// TIA Portal project "HydroPlantProject" (V15)

(* hardware
DEVICE "S71500/ET200MP station_1"  S7-1500 station
   slot 0: "Rail_0"  Rack  6ES7 590-1***0-0AA0
   slot 1: "PLC_1"  CPU 1511-1 PN  6ES7 511-1AK00-0AB0  V1.8
      slot 3: "CPU display_1"  6ES7591-1AA00-0AA0
DEVICE "PC-System_1"  SIMATIC PC station
   slot 0: "SIMATIC PC station"  Rail  SIMATIC PC-Station  V1.0
      slot 125: "Stationmanager"  Station_Manager  V6.0.4
   slot 1: "HMI_RT_1"  WinCC RT Advanced  6AV2 104-0xxxx-xxxx  15.0.0.0
      slot 33792: "Host interface"  Host interface
   slot 2: "IE general_1"  IE General  IE_CP  V8.2.0
*)

// ===== PLC "PLC_1"  CPU 1511-1 PN =====

VAR_GLOBAL   // PLC tag table "Default tag table"
   "Brake_Out" AT %M0.0 : Bool;
   "Baffle_Out" AT %MW18 : Int;
   "RPM_In" AT %MW2 : Int;
   "OilTemp_In" AT %MW4 : Int;
   "OilPumpVFDen_Out" AT %M0.1 : Bool;
   "OilPumpVFDsp_Out" AT %MW6 : Int;
   "OilFlow_In" AT %MW8 : Int;
   "Current_In" AT %MW10 : Int;
   "Baffle_En" AT %M0.2 : Bool;
   "ProgLang" AT %MW12 : Int;
   "ONS1" AT %M0.3 : Bool;
   "PB_LAD" AT %M0.4 : Bool;
   "ONS" AT %M0.5 : Bool;
   "PB_FBD" AT %M0.6 : Bool;
   "PB_SCL" AT %M0.7 : Bool;
   "PB_STL" AT %M1.0 : Bool;
   "ONS2" AT %M1.1 : Bool;
   "ONS3" AT %M1.2 : Bool;
   "ONS4" AT %M1.3 : Bool;
   "AlarmHorn_Out" AT %M1.4 : Bool;
   "Stationinterlock_Out" AT %M1.5 : Bool;
   "OilPumpVFDpct" AT %MW14 : Int;
   "BafflePct" AT %MW16 : Int;
   "OilTemp" AT %MW20 : Int;
   "OilFlow" AT %MW24 : Int;
   "RPM" AT %MW26 : Int;
   "Current" AT %MW28 : Int;
   "OilPumpVFDhand_Pb" AT %M1.6 : Bool;
   "OilPumpVFDoff_Pb" AT %M1.7 : Bool;
   "OilPumpVFDauto_Pb" AT %M22.0 : Bool;
   "OilPumpVFDhoa" AT %MW30 : Int;
   "BrakeHoa" AT %MW32 : Int;
   "BrakeOff_Pb" AT %M22.1 : Bool;
   "BrakeHand_Pb" AT %M22.2 : Bool;
   "BrakeAuto_Pb" AT %M22.3 : Bool;
   "AlarmHornOff_Pb" AT %M22.4 : Bool;
   "AlarmHornHand_Pb" AT %M22.5 : Bool;
   "AlarmHornHoa" AT %MW34 : Int;
   "AlarmHornAuto_Pb" AT %M22.6 : Bool;
   "StationintOff_Pb" AT %M22.7 : Bool;
   "StationintHand_Pb" AT %M23.0 : Bool;
   "StationintAuto_Pb" AT %M23.1 : Bool;
   "StationintHoa" AT %MW36 : Int;
   "OilPumpVFD_Ctrl" AT %M23.2 : Bool;
   "Bracke_Ctrl" AT %M23.3 : Bool;
   "ALarmHorn_Ctrl" AT %M23.4 : Bool;
   "Stationint_Ctrl" AT %M23.5 : Bool;
   "OilLowFlowDelay_Sp" AT %MW38 : Int;
   "AlarmReset" AT %M23.6 : Bool;
   "AlarmSilence" AT %M23.7 : Bool;
   "OilLowFlowAlarm" AT %M40.0 : Bool;
   "OilLowFlowNotify" AT %M40.1 : Bool;
   "OilLLFlow_Sp" AT %MW42 : Int;
   "OverCurrent_Sp" AT %MW44 : Int;
   "OverCurrentAlarm" AT %M40.2 : Bool;
   "OverCurrentAlarm(1)" AT %M40.3 : Bool;
   "OverCurrentNotify" AT %M40.4 : Bool;
   "OverCurrentDelay_Sp" AT %MW46 : Int;
   "HighoilTepDelay_Sp" AT %MW48 : Int;
   "HighOilTemp _Sp" AT %MW50 : Int;
   "OilTempAlarm" AT %M40.5 : Bool;
   "OilTempAlarmNotify" AT %M40.6 : Bool;
   "RottorOverspeed_Sp" AT %MW52 : Int;
   "RottorOverspeedDelay_Sp" AT %MW54 : Int;
   "RottorOverspeedAlarm" AT %M40.7 : Bool;
   "RottorOverspeedNotify" AT %M41.0 : Bool;
   "OilHighFlowAlarm" AT %M41.1 : Bool;
   "OilHighFlowNotify" AT %M41.2 : Bool;
   "OilHighFlowDelay_Sp" AT %MW56 : Int;
   "OilHHFlow_Sp" AT %MW58 : Int;
   "BraheFailuerDelay_Sp" AT %MW60 : Int;
   "BrakeFalierAlarm" AT %M41.3 : Bool;
   "BrakeFalierAlarmNotify" AT %M41.4 : Bool;
   "EStop" AT %M41.5 : Bool;
   "ESTOPAlarm" AT %M41.6 : Bool;
   "EStapAlarmNotify" AT %M41.7 : Bool;
   "Tag_1" AT %T1 : Timer;
   "WarmupMode" AT %M62.0 : Bool;
   "StabilizeMode" AT %M62.1 : Bool;
   "GenerationMode" AT %M62.2 : Bool;
   "CooldownMode" AT %M62.3 : Bool;
   "IdleMode" AT %M62.4 : Bool;
   "FaultMode" AT %M62.5 : Bool;
   "SystemSTART_Pb" AT %M62.6 : Bool;
   "WarmupRPM" AT %MW63 : Int;
   "RPM_SP" AT %MW64 : Int;
   "BaffleHOA" AT %MW66 : Int;
   "Baffle_Ctrl" AT %M62.7 : Bool;
   "WarmupVFDpct" AT %MW68 : Int;
   "VFD_sp" AT %MW70 : Int;
   "WarmupOILTemp" AT %MW72 : Int;
   "WarmupOilTempDelay_sp" AT %MW74 : Int;
   "WarmupTransition" AT %M76.0 : Bool;
   "BafflePIDsp" AT %MW78 : Int;
   "StabilizeKWsp" AT %MW80 : Int;
   "StabilizeDelay_sp" AT %MW82 : Int;
   "StabilizeTranzition" AT %M76.1 : Bool;
   "STARTSequnceBIT" AT %M76.2 : Bool;
   "SystemSTOP_PB" AT %M76.3 : Bool;
   "GenerationTransition" AT %M76.4 : Bool;
   "BafflePIDin" AT %MW84 : Int;
   "CooldownRPM" AT %MW86 : Int;
   "CooldownDelay_Sp" AT %MW88 : Int;
   "CooldawnTransition" AT %M76.5 : Bool;
   "CoolDownRPM_sp" AT %MW90 : Int;
   "CoolDownOilTemp_sp" AT %MW92 : Int;
   "SequenceRunning" AT %M76.6 : Bool;
   "ONS5" AT %M76.7 : Bool;
   "StabilizeTransition" AT %M77.0 : Bool;
END_VAR

DATA_BLOCK "SimLogic_DB"   // DB1
{ S7_Optimized_Access := 'TRUE' }
VERSION : 0.1
// stored: InstanceOfName SimLogic
"SimLogic"
BEGIN
END_DATA_BLOCK

DATA_BLOCK "SimLogic_DB_1"   // DB2
{ S7_Optimized_Access := 'TRUE' }
VERSION : 0.1
// stored: InstanceOfName SimLogic
"SimLogic"
BEGIN
END_DATA_BLOCK

DATA_BLOCK "IO_LAD_DB"   // DB4
{ S7_Optimized_Access := 'TRUE' }
VERSION : 0.1
// stored: InstanceOfName IO_LAD
"IO_LAD"
BEGIN
END_DATA_BLOCK

DATA_BLOCK "IO_FBD_DB"   // DB5
{ S7_Optimized_Access := 'TRUE' }
VERSION : 0.1
// stored: InstanceOfName IO_FBD
"IO_FBD"
BEGIN
END_DATA_BLOCK

DATA_BLOCK "IO_SCL_DB"   // DB6
{ S7_Optimized_Access := 'TRUE' }
VERSION : 0.1
// stored: InstanceOfName IO_SCL
"IO_SCL"
BEGIN
END_DATA_BLOCK

DATA_BLOCK "IO_STL_DB"   // DB7
{ S7_Optimized_Access := 'TRUE' }
VERSION : 0.1
// stored: InstanceOfName IO_STL
"IO_STL"
BEGIN
END_DATA_BLOCK

DATA_BLOCK "ALARMS_LAD_DB"   // DB8
{ S7_Optimized_Access := 'TRUE' }
VERSION : 0.1
// stored: InstanceOfName ALARMS_LAD
"ALARMS_LAD"
BEGIN
END_DATA_BLOCK

DATA_BLOCK "SCP_DB"   // DB9
{ S7_Optimized_Access := 'TRUE' }
VERSION : 0.1
// stored: InstanceOfName SCP
"SCP"
BEGIN
END_DATA_BLOCK

DATA_BLOCK "SCP_DB_1"   // DB10
{ S7_Optimized_Access := 'TRUE' }
VERSION : 0.1
// stored: InstanceOfName SCP
"SCP"
BEGIN
END_DATA_BLOCK

DATA_BLOCK "HOA_LAD_DB"   // DB11
{ S7_Optimized_Access := 'TRUE' }
VERSION : 0.1
// stored: InstanceOfName HOA_LAD
"HOA_LAD"
BEGIN
END_DATA_BLOCK

DATA_BLOCK "HOA_FBD_DB"   // DB12
{ S7_Optimized_Access := 'TRUE' }
VERSION : 0.1
// stored: InstanceOfName HOA_FBD
"HOA_FBD"
BEGIN
END_DATA_BLOCK

DATA_BLOCK "HOA_SCL_DB"   // DB13
{ S7_Optimized_Access := 'TRUE' }
VERSION : 0.1
// stored: InstanceOfName HOA_SCL
"HOA_SCL"
BEGIN
END_DATA_BLOCK

DATA_BLOCK "HOA_STL_DB"   // DB14
{ S7_Optimized_Access := 'TRUE' }
VERSION : 0.1
// stored: InstanceOfName HOA_STL
"HOA_STL"
BEGIN
END_DATA_BLOCK

DATA_BLOCK "ALARMS_FBD_DB"   // DB15
{ S7_Optimized_Access := 'TRUE' }
VERSION : 0.1
// stored: InstanceOfName ALARMS_FBD
"ALARMS_FBD"
BEGIN
END_DATA_BLOCK

DATA_BLOCK "ALARMS_SCL_DB"   // DB16
{ S7_Optimized_Access := 'TRUE' }
VERSION : 0.1
// stored: InstanceOfName ALARMS_SCL
"ALARMS_SCL"
BEGIN
END_DATA_BLOCK

DATA_BLOCK "ALARMS_STL_DB"   // DB18
{ S7_Optimized_Access := 'TRUE' }
VERSION : 0.1
// stored: InstanceOfName ALARMS_STL
"ALARMS_STL"
BEGIN
END_DATA_BLOCK

DATA_BLOCK "SEQUENCE_DB"   // DB37
{ S7_Optimized_Access := 'TRUE' }
VERSION : 0.1
// stored: InstanceOfName SEQUENCE
"SEQUENCE"
BEGIN
END_DATA_BLOCK

// folder: System blocks/Program resources

DATA_BLOCK "IEC_Timer_0_DB_25"   // DB3
{ S7_Optimized_Access := 'TRUE' }
AUTHOR : Simatic
FAMILY : IEC
NAME : IEC_TMR
VERSION : 1.0
// stored: InstanceOfName IEC_TIMER
"IEC_TIMER"
BEGIN
END_DATA_BLOCK

DATA_BLOCK "IEC_Timer_0_DB"   // DB17
{ S7_Optimized_Access := 'TRUE' }
AUTHOR : Simatic
FAMILY : IEC
NAME : IEC_TMR
VERSION : 1.0
// stored: InstanceOfName IEC_TIMER
"IEC_TIMER"
BEGIN
END_DATA_BLOCK

DATA_BLOCK "IEC_Timer_0_DB_1"   // DB19
{ S7_Optimized_Access := 'TRUE' }
AUTHOR : Simatic
FAMILY : IEC
NAME : IEC_TMR
VERSION : 1.0
// stored: InstanceOfName IEC_TIMER
"IEC_TIMER"
BEGIN
END_DATA_BLOCK

DATA_BLOCK "IEC_Timer_0_DB_2"   // DB20
{ S7_Optimized_Access := 'TRUE' }
AUTHOR : Simatic
FAMILY : IEC
NAME : IEC_TMR
VERSION : 1.0
// stored: InstanceOfName IEC_TIMER
"IEC_TIMER"
BEGIN
END_DATA_BLOCK

DATA_BLOCK "IEC_Timer_0_DB_3"   // DB21
{ S7_Optimized_Access := 'TRUE' }
AUTHOR : Simatic
FAMILY : IEC
NAME : IEC_TMR
VERSION : 1.0
// stored: InstanceOfName IEC_TIMER
"IEC_TIMER"
BEGIN
END_DATA_BLOCK

DATA_BLOCK "IEC_Timer_0_DB_4"   // DB22
{ S7_Optimized_Access := 'TRUE' }
AUTHOR : Simatic
FAMILY : IEC
NAME : IEC_TMR
VERSION : 1.0
// stored: InstanceOfName IEC_TIMER
"IEC_TIMER"
BEGIN
END_DATA_BLOCK

DATA_BLOCK "IEC_Timer_0_DB_5"   // DB23
{ S7_Optimized_Access := 'TRUE' }
AUTHOR : Simatic
FAMILY : IEC
NAME : IEC_TMR
VERSION : 1.0
// stored: InstanceOfName IEC_TIMER
"IEC_TIMER"
BEGIN
END_DATA_BLOCK

DATA_BLOCK "IEC_Timer_0_DB_6"   // DB24
{ S7_Optimized_Access := 'TRUE' }
AUTHOR : Simatic
FAMILY : IEC
NAME : IEC_TMR
VERSION : 1.0
// stored: InstanceOfName IEC_TIMER
"IEC_TIMER"
BEGIN
END_DATA_BLOCK

DATA_BLOCK "IEC_Timer_0_DB_7"   // DB25
{ S7_Optimized_Access := 'TRUE' }
AUTHOR : Simatic
FAMILY : IEC
NAME : IEC_TMR
VERSION : 1.0
// stored: InstanceOfName IEC_TIMER
"IEC_TIMER"
BEGIN
END_DATA_BLOCK

DATA_BLOCK "IEC_Timer_0_DB_8"   // DB26
{ S7_Optimized_Access := 'TRUE' }
AUTHOR : Simatic
FAMILY : IEC
NAME : IEC_TMR
VERSION : 1.0
// stored: InstanceOfName IEC_TIMER
"IEC_TIMER"
BEGIN
END_DATA_BLOCK

DATA_BLOCK "IEC_Timer_0_DB_9"   // DB27
{ S7_Optimized_Access := 'TRUE' }
AUTHOR : Simatic
FAMILY : IEC
NAME : IEC_TMR
VERSION : 1.0
// stored: InstanceOfName IEC_TIMER
"IEC_TIMER"
BEGIN
END_DATA_BLOCK

DATA_BLOCK "IEC_Timer_0_DB_10"   // DB28
{ S7_Optimized_Access := 'TRUE' }
AUTHOR : Simatic
FAMILY : IEC
NAME : IEC_TMR
VERSION : 1.0
// stored: InstanceOfName IEC_TIMER
"IEC_TIMER"
BEGIN
END_DATA_BLOCK

DATA_BLOCK "IEC_Timer_0_DB_11"   // DB29
{ S7_Optimized_Access := 'TRUE' }
AUTHOR : Simatic
FAMILY : IEC
NAME : IEC_TMR
VERSION : 1.0
// stored: InstanceOfName IEC_TIMER
"IEC_TIMER"
BEGIN
END_DATA_BLOCK

DATA_BLOCK "IEC_Timer_0_DB_12"   // DB30
{ S7_Optimized_Access := 'TRUE' }
AUTHOR : Simatic
FAMILY : IEC
NAME : IEC_TMR
VERSION : 1.0
// stored: InstanceOfName IEC_TIMER
"IEC_TIMER"
BEGIN
END_DATA_BLOCK

DATA_BLOCK "IEC_Timer_0_DB_13"   // DB31
{ S7_Optimized_Access := 'TRUE' }
AUTHOR : Simatic
FAMILY : IEC
NAME : IEC_TMR
VERSION : 1.0
// stored: InstanceOfName IEC_TIMER
"IEC_TIMER"
BEGIN
END_DATA_BLOCK

DATA_BLOCK "IEC_Timer_0_DB_14"   // DB32
{ S7_Optimized_Access := 'TRUE' }
AUTHOR : Simatic
FAMILY : IEC
NAME : IEC_TMR
VERSION : 1.0
// stored: InstanceOfName IEC_TIMER
"IEC_TIMER"
BEGIN
END_DATA_BLOCK

DATA_BLOCK "IEC_Timer_0_DB_15"   // DB33
{ S7_Optimized_Access := 'TRUE' }
AUTHOR : Simatic
FAMILY : IEC
NAME : IEC_TMR
VERSION : 1.0
// stored: InstanceOfName IEC_TIMER
"IEC_TIMER"
BEGIN
END_DATA_BLOCK

DATA_BLOCK "IEC_Timer_0_DB_16"   // DB34
{ S7_Optimized_Access := 'TRUE' }
AUTHOR : Simatic
FAMILY : IEC
NAME : IEC_TMR
VERSION : 1.0
// stored: InstanceOfName IEC_TIMER
"IEC_TIMER"
BEGIN
END_DATA_BLOCK

DATA_BLOCK "IEC_Timer_0_DB_17"   // DB35
{ S7_Optimized_Access := 'TRUE' }
AUTHOR : Simatic
FAMILY : IEC
NAME : IEC_TMR
VERSION : 1.0
// stored: InstanceOfName IEC_TIMER
"IEC_TIMER"
BEGIN
END_DATA_BLOCK

DATA_BLOCK "IEC_Timer_0_DB_18"   // DB36
{ S7_Optimized_Access := 'TRUE' }
AUTHOR : Simatic
FAMILY : IEC
NAME : IEC_TMR
VERSION : 1.0
// stored: InstanceOfName IEC_TIMER
"IEC_TIMER"
BEGIN
END_DATA_BLOCK

DATA_BLOCK "IEC_Timer_0_DB_19"   // DB38
{ S7_Optimized_Access := 'TRUE' }
AUTHOR : Simatic
FAMILY : IEC
NAME : IEC_TMR
VERSION : 1.0
// stored: InstanceOfName IEC_TIMER
"IEC_TIMER"
BEGIN
END_DATA_BLOCK

DATA_BLOCK "IEC_Timer_0_DB_20"   // DB39
{ S7_Optimized_Access := 'TRUE' }
AUTHOR : Simatic
FAMILY : IEC
NAME : IEC_TMR
VERSION : 1.0
// stored: InstanceOfName IEC_TIMER
"IEC_TIMER"
BEGIN
END_DATA_BLOCK

DATA_BLOCK "IEC_Timer_0_DB_30"   // DB40
{ S7_Optimized_Access := 'TRUE' }
AUTHOR : Simatic
FAMILY : IEC
NAME : IEC_TMR
VERSION : 1.0
// stored: InstanceOfName IEC_TIMER
"IEC_TIMER"
BEGIN
END_DATA_BLOCK

DATA_BLOCK "IEC_Timer_0_DB_21"   // DB41
{ S7_Optimized_Access := 'TRUE' }
AUTHOR : Simatic
FAMILY : IEC
NAME : IEC_TMR
VERSION : 1.0
// stored: InstanceOfName IEC_TIMER
"IEC_TIMER"
BEGIN
END_DATA_BLOCK

DATA_BLOCK "IEC_Timer_1_DB"   // DB43
{ S7_Optimized_Access := 'TRUE' }
AUTHOR : Simatic
FAMILY : IEC
NAME : IEC_TMR
VERSION : 1.0
// stored: InstanceOfName IEC_TIMER
"IEC_TIMER"
BEGIN
END_DATA_BLOCK

DATA_BLOCK "IEC_Timer_0_DB_22"   // DB44
{ S7_Optimized_Access := 'TRUE' }
AUTHOR : Simatic
FAMILY : IEC
NAME : IEC_TMR
VERSION : 1.0
// stored: InstanceOfName IEC_TIMER
"IEC_TIMER"
BEGIN
END_DATA_BLOCK

DATA_BLOCK "IEC_Timer_0_DB_23"   // DB45
{ S7_Optimized_Access := 'TRUE' }
AUTHOR : Simatic
FAMILY : IEC
NAME : IEC_TMR
VERSION : 1.0
// stored: InstanceOfName IEC_TIMER
"IEC_TIMER"
BEGIN
END_DATA_BLOCK

DATA_BLOCK "IEC_Timer_0_DB_24"   // DB46
{ S7_Optimized_Access := 'TRUE' }
AUTHOR : Simatic
FAMILY : IEC
NAME : IEC_TMR
VERSION : 1.0
// stored: InstanceOfName IEC_TIMER
"IEC_TIMER"
BEGIN
END_DATA_BLOCK

DATA_BLOCK "IEC_Timer_0_DB_26"   // DB47
{ S7_Optimized_Access := 'TRUE' }
AUTHOR : Simatic
FAMILY : IEC
NAME : IEC_TMR
VERSION : 1.0
// stored: InstanceOfName IEC_TIMER
"IEC_TIMER"
BEGIN
END_DATA_BLOCK

DATA_BLOCK "IEC_Timer_0_DB_27"   // DB48
{ S7_Optimized_Access := 'TRUE' }
AUTHOR : Simatic
FAMILY : IEC
NAME : IEC_TMR
VERSION : 1.0
// stored: InstanceOfName IEC_TIMER
"IEC_TIMER"
BEGIN
END_DATA_BLOCK

// folder: (top level)

FUNCTION_BLOCK "SimLogic"   // FB1, FBD
{ S7_Optimized_Access := 'TRUE' }
VERSION : 0.1
   VAR
      "TO" : Bool;
      rpmv : Int;
      addrpmv : Bool;
      otsp : Int;
      ott : Int;
      TO1 : Bool;
      TO2 : Bool;
      be2 : Int;
      be3 : Int;
      be1 : Int;
      TO3 : Bool;
   END_VAR
   VAR_TEMP
      bf : Int;
      rpmvt : Int;
      bfr : Real;
   END_VAR
BEGIN

REGION Network 1
   // RPM
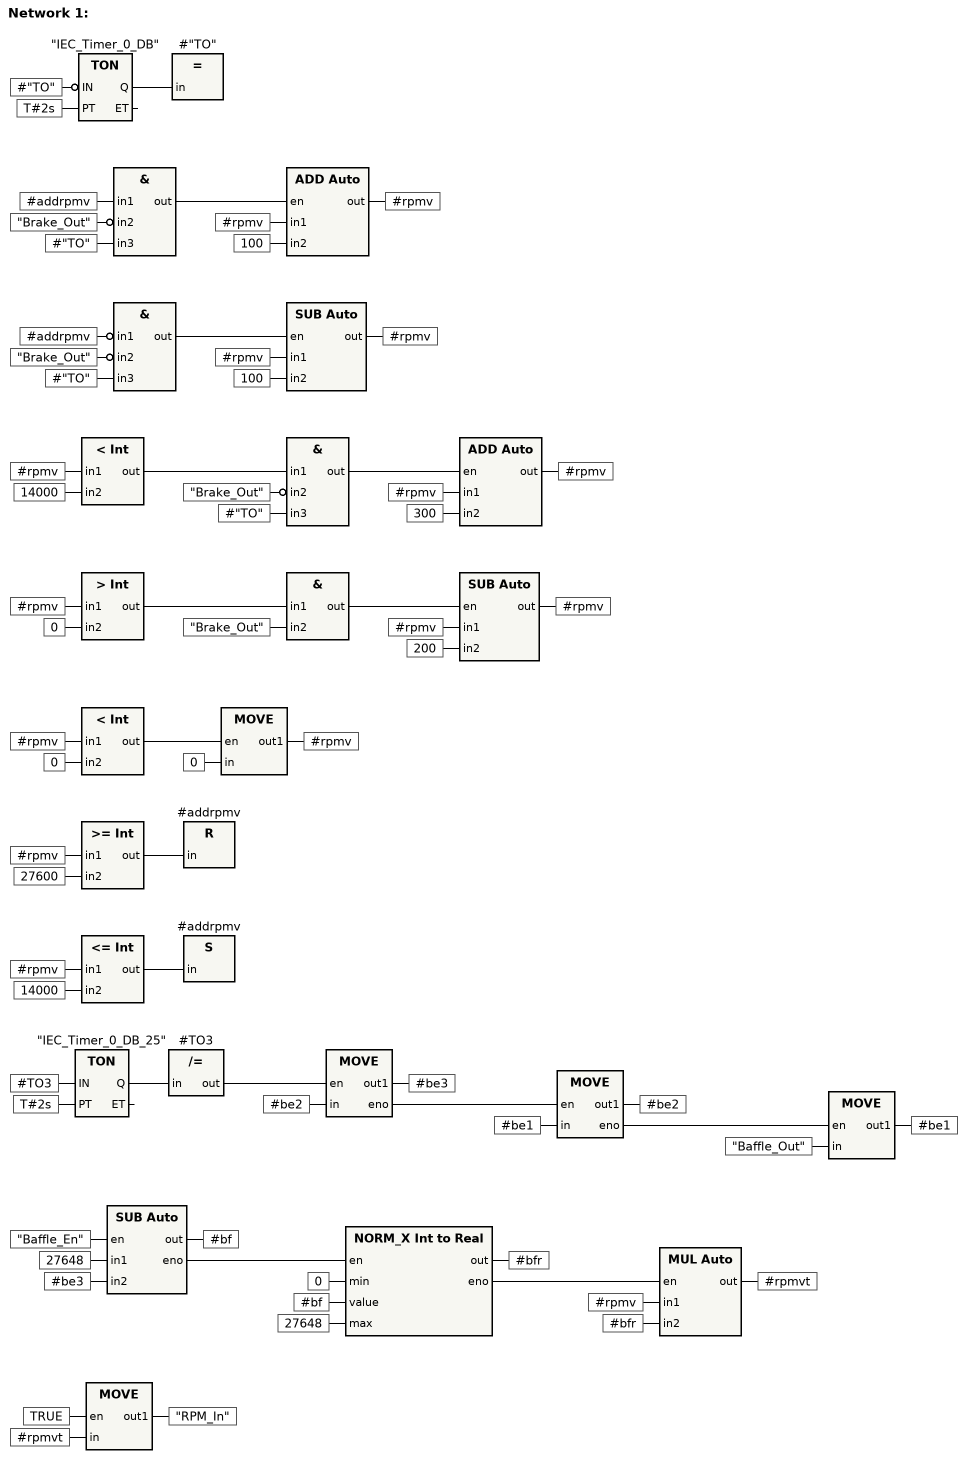
   "IEC_Timer_0_DB".TON(IN := NOT #"TO", PT := T#2s);
   #"TO" := "IEC_Timer_0_DB".Q;
   IF #addrpmv AND NOT "Brake_Out" AND #"TO" THEN #rpmv := #rpmv + 100; END_IF;
   IF NOT #addrpmv AND NOT "Brake_Out" AND #"TO" THEN #rpmv := #rpmv - 100; END_IF;
   IF (#rpmv < 14000) AND NOT "Brake_Out" AND #"TO" THEN #rpmv := #rpmv + 300; END_IF;
   IF (#rpmv > 0) AND "Brake_Out" THEN #rpmv := #rpmv - 200; END_IF;
   IF #rpmv < 0 THEN #rpmv := 0; END_IF;
   IF #rpmv >= 27600 THEN #addrpmv := FALSE; END_IF;
   IF #rpmv <= 14000 THEN #addrpmv := TRUE; END_IF;
   "IEC_Timer_0_DB_25".TON(IN := #TO3, PT := T#2s);
   #TO3 := NOT "IEC_Timer_0_DB_25".Q;
   IF "IEC_Timer_0_DB_25".Q THEN
       #be3 := #be2;
       #be2 := #be1;
       #be1 := "Baffle_Out";
   END_IF;
   IF "Baffle_En" THEN
       #bf := 27648 - #be3;
       #bfr := NORM_X(MIN := 0, VALUE := #bf, MAX := 27648);
       #rpmvt := #rpmv * #bfr;
   END_IF;
   IF TRUE THEN "RPM_In" := #rpmvt; END_IF;
END_REGION

REGION Network 2
   // Oil Temp
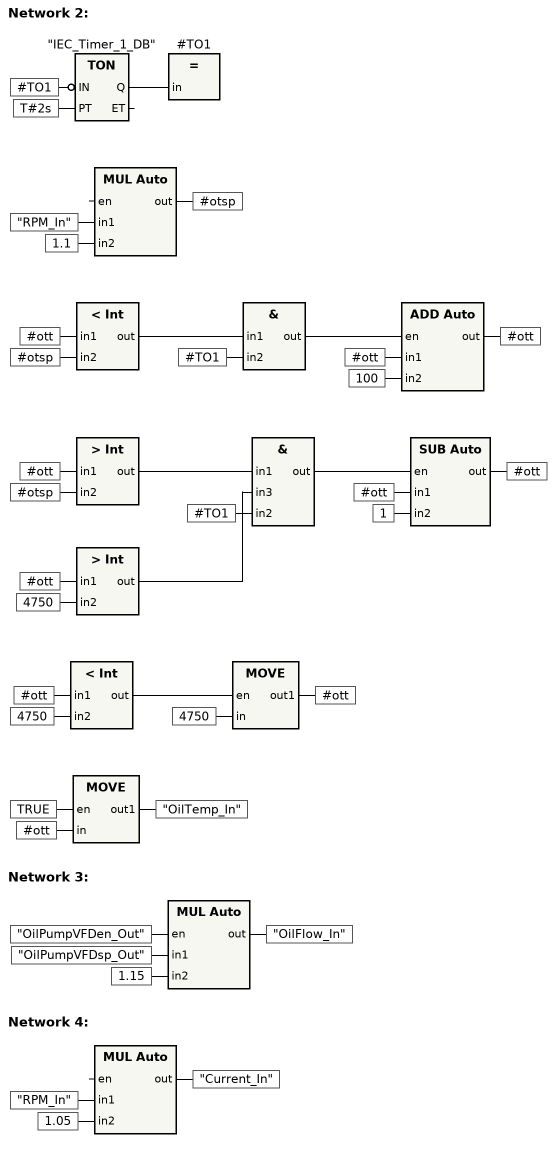
   "IEC_Timer_1_DB".TON(IN := NOT #TO1, PT := T#2s);
   #TO1 := "IEC_Timer_1_DB".Q;
   #otsp := "RPM_In" * 1.1;
   IF (#ott < #otsp) AND #TO1 THEN #ott := #ott + 100; END_IF;
   IF (#ott > #otsp) AND (#ott > 4750) AND #TO1 THEN #ott := #ott - 1; END_IF;
   IF #ott < 4750 THEN #ott := 4750; END_IF;
   IF TRUE THEN "OilTemp_In" := #ott; END_IF;
END_REGION

REGION Network 3
   // Oil Flow
   IF "OilPumpVFDen_Out" THEN "OilFlow_In" := "OilPumpVFDsp_Out" * 1.15; END_IF;
END_REGION

REGION Network 4
   // Current
   "Current_In" := "RPM_In" * 1.05;
END_REGION
END_FUNCTION_BLOCK

FUNCTION_BLOCK "IO_LAD"   // FB2, LAD
{ S7_Optimized_Access := 'TRUE' }
VERSION : 0.1
BEGIN

REGION Network 1
   // Digital Output
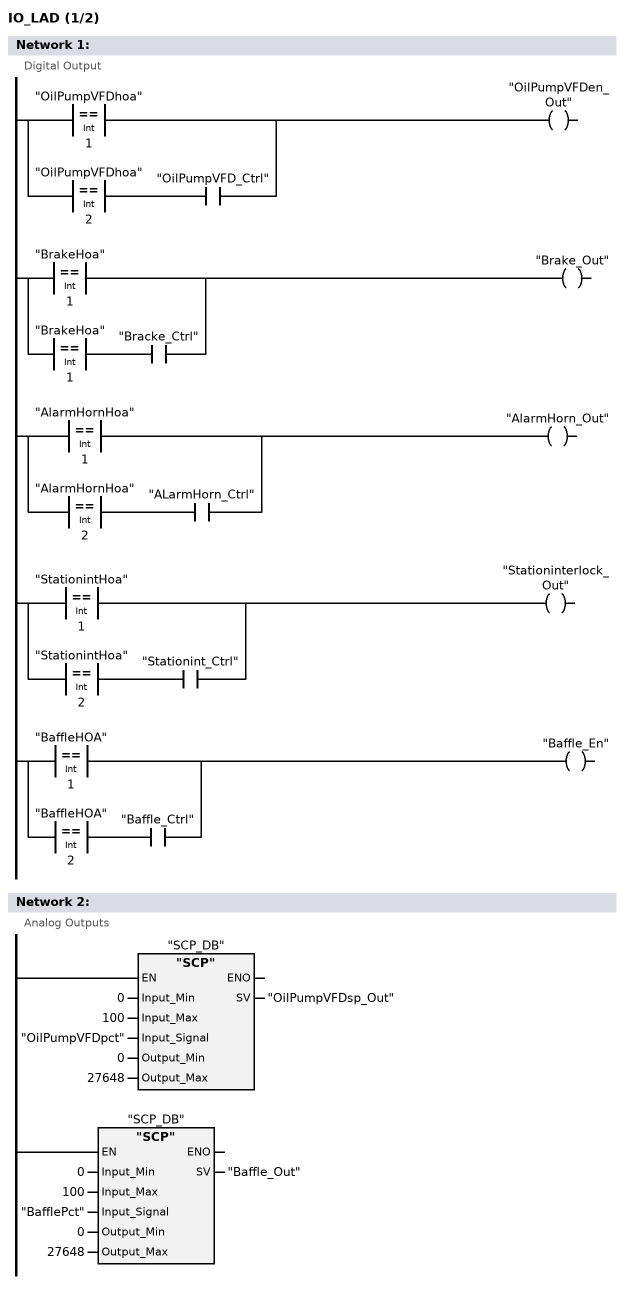
   RUNG wire#powerrail
      { S7_Templates := "SrcType := Int" } EQ_Contact(in1 := "OilPumpVFDhoa", in2 := 1)
      wire#w1
      Coil( "OilPumpVFDen_Out" )
   END_RUNG
   RUNG wire#powerrail
      { S7_Templates := "SrcType := Int" } EQ_Contact(in1 := "OilPumpVFDhoa", in2 := 2)
      Contact( "OilPumpVFD_Ctrl" )
   END_RUNG wire#w1
   RUNG wire#powerrail
      { S7_Templates := "SrcType := Int" } EQ_Contact(in1 := "BrakeHoa", in2 := 1)
      wire#w2
      Coil( "Brake_Out" )
   END_RUNG
   RUNG wire#powerrail
      { S7_Templates := "SrcType := Int" } EQ_Contact(in1 := "BrakeHoa", in2 := 1)
      Contact( "Bracke_Ctrl" )
   END_RUNG wire#w2
   RUNG wire#powerrail
      { S7_Templates := "SrcType := Int" } EQ_Contact(in1 := "AlarmHornHoa", in2 := 1)
      wire#w3
      Coil( "AlarmHorn_Out" )
   END_RUNG
   RUNG wire#powerrail
      { S7_Templates := "SrcType := Int" } EQ_Contact(in1 := "AlarmHornHoa", in2 := 2)
      Contact( "ALarmHorn_Ctrl" )
   END_RUNG wire#w3
   RUNG wire#powerrail
      { S7_Templates := "SrcType := Int" } EQ_Contact(in1 := "StationintHoa", in2 := 1)
      wire#w4
      Coil( "Stationinterlock_Out" )
   END_RUNG
   RUNG wire#powerrail
      { S7_Templates := "SrcType := Int" } EQ_Contact(in1 := "StationintHoa", in2 := 2)
      Contact( "Stationint_Ctrl" )
   END_RUNG wire#w4
   RUNG wire#powerrail
      { S7_Templates := "SrcType := Int" } EQ_Contact(in1 := "BaffleHOA", in2 := 1)
      wire#w5
      Coil( "Baffle_En" )
   END_RUNG
   RUNG wire#powerrail
      { S7_Templates := "SrcType := Int" } EQ_Contact(in1 := "BaffleHOA", in2 := 2)
      Contact( "Baffle_Ctrl" )
   END_RUNG wire#w5
   // the same network as SCL:
   "OilPumpVFDen_Out" := ("OilPumpVFDhoa" = 1) OR (("OilPumpVFDhoa" = 2) AND "OilPumpVFD_Ctrl");
   "Brake_Out" := ("BrakeHoa" = 1) OR (("BrakeHoa" = 1) AND "Bracke_Ctrl");
   "AlarmHorn_Out" := ("AlarmHornHoa" = 1) OR (("AlarmHornHoa" = 2) AND "ALarmHorn_Ctrl");
   "Stationinterlock_Out" := ("StationintHoa" = 1) OR (("StationintHoa" = 2) AND "Stationint_Ctrl");
   "Baffle_En" := ("BaffleHOA" = 1) OR (("BaffleHOA" = 2) AND "Baffle_Ctrl");
END_REGION

REGION Network 2
   // Analog Outputs
   RUNG wire#powerrail
      "SCP_DB"(Input_Min := 0, Input_Max := 100, Input_Signal := "OilPumpVFDpct", Output_Min := 0, Output_Max := 27648, SV => "OilPumpVFDsp_Out")
   END_RUNG
   RUNG wire#powerrail
      "SCP_DB"(Input_Min := 0, Input_Max := 100, Input_Signal := "BafflePct", Output_Min := 0, Output_Max := 27648, SV => "Baffle_Out")
   END_RUNG
   // the same network as SCL:
   "SCP_DB"(Input_Min := 0,   // "SCP"
            Input_Max := 100,
            Input_Signal := "OilPumpVFDpct",
            Output_Min := 0,
            Output_Max := 27648,
            SV => "OilPumpVFDsp_Out");
   "SCP_DB"(Input_Min := 0,   // "SCP"
            Input_Max := 100,
            Input_Signal := "BafflePct",
            Output_Min := 0,
            Output_Max := 27648,
            SV => "Baffle_Out");
END_REGION

REGION Network 3
   // Analog Inputs
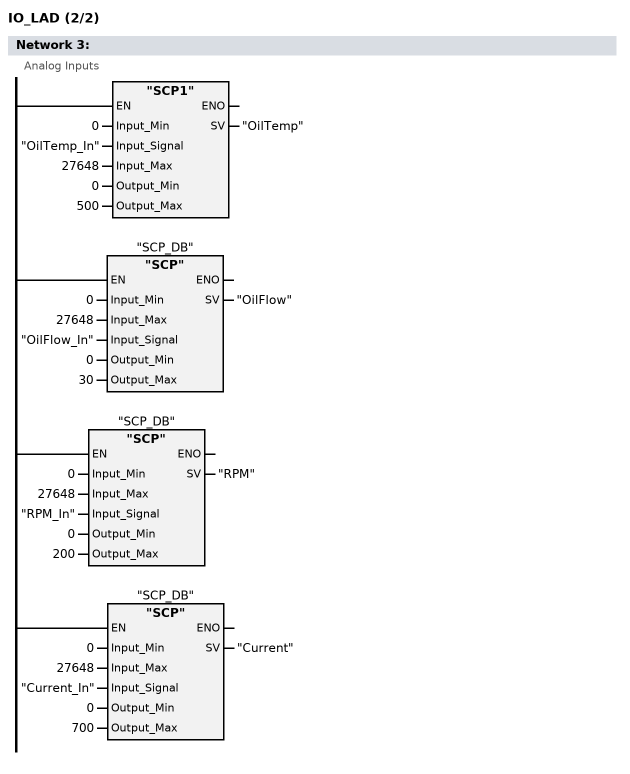
   RUNG wire#powerrail
      "SCP1"(Input_Min := 0, Input_Signal := "OilTemp_In", Input_Max := 27648, Output_Min := 0, Output_Max := 500, SV => "OilTemp")
   END_RUNG
   RUNG wire#powerrail
      "SCP_DB"(Input_Min := 0, Input_Max := 27648, Input_Signal := "OilFlow_In", Output_Min := 0, Output_Max := 30, SV => "OilFlow")
   END_RUNG
   RUNG wire#powerrail
      "SCP_DB"(Input_Min := 0, Input_Max := 27648, Input_Signal := "RPM_In", Output_Min := 0, Output_Max := 200, SV => "RPM")
   END_RUNG
   RUNG wire#powerrail
      "SCP_DB"(Input_Min := 0, Input_Max := 27648, Input_Signal := "Current_In", Output_Min := 0, Output_Max := 700, SV => "Current")
   END_RUNG
   // the same network as SCL:
   "SCP1"(Input_Min := 0,
          Input_Signal := "OilTemp_In",
          Input_Max := 27648,
          Output_Min := 0,
          Output_Max := 500,
          SV => "OilTemp");
   "SCP_DB"(Input_Min := 0,   // "SCP"
            Input_Max := 27648,
            Input_Signal := "OilFlow_In",
            Output_Min := 0,
            Output_Max := 30,
            SV => "OilFlow");
   "SCP_DB"(Input_Min := 0,   // "SCP"
            Input_Max := 27648,
            Input_Signal := "RPM_In",
            Output_Min := 0,
            Output_Max := 200,
            SV => "RPM");
   "SCP_DB"(Input_Min := 0,   // "SCP"
            Input_Max := 27648,
            Input_Signal := "Current_In",
            Output_Min := 0,
            Output_Max := 700,
            SV => "Current");
END_REGION
END_FUNCTION_BLOCK

FUNCTION_BLOCK "IO_FBD"   // FB3, FBD
{ S7_Optimized_Access := 'TRUE' }
VERSION : 0.1
   VAR_TEMP
      tv : Real;
   END_VAR
BEGIN

REGION Network 1
   // Digital Outputs
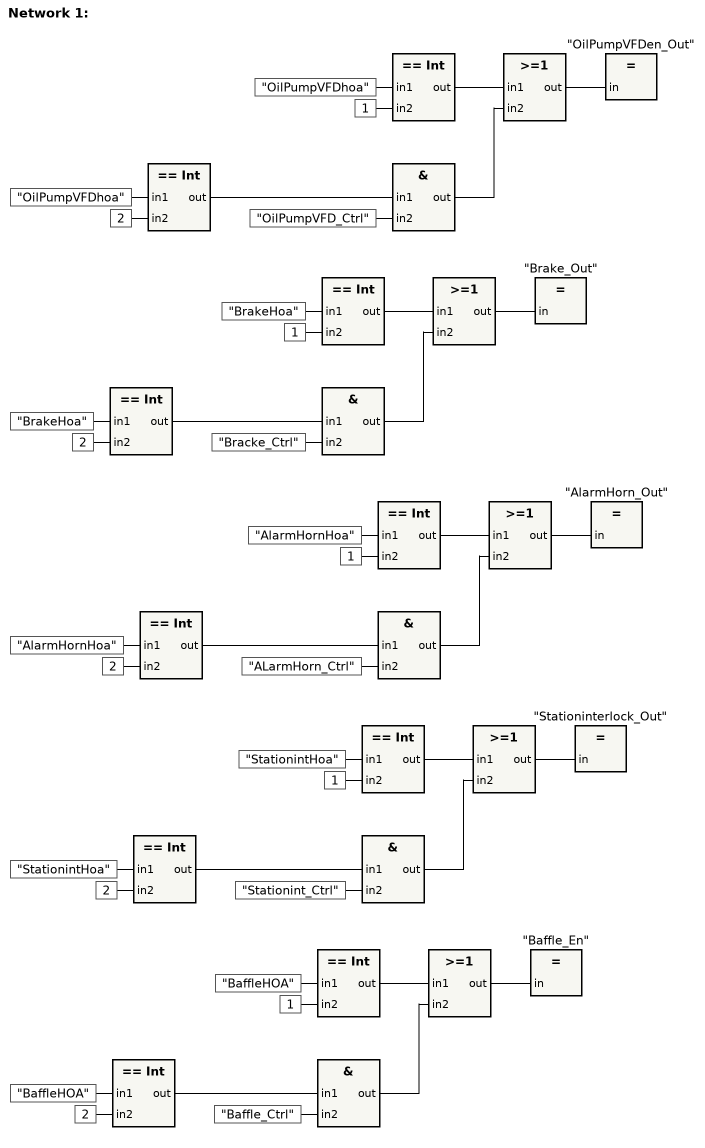
   "OilPumpVFDen_Out" := ("OilPumpVFDhoa" = 1) OR (("OilPumpVFDhoa" = 2) AND "OilPumpVFD_Ctrl");
   "Brake_Out" := ("BrakeHoa" = 1) OR (("BrakeHoa" = 2) AND "Bracke_Ctrl");
   "AlarmHorn_Out" := ("AlarmHornHoa" = 1) OR (("AlarmHornHoa" = 2) AND "ALarmHorn_Ctrl");
   "Stationinterlock_Out" := ("StationintHoa" = 1) OR (("StationintHoa" = 2) AND "Stationint_Ctrl");
   "Baffle_En" := ("BaffleHOA" = 1) OR (("BaffleHOA" = 2) AND "Baffle_Ctrl");
END_REGION

REGION Network 2
   // Analog Outputs
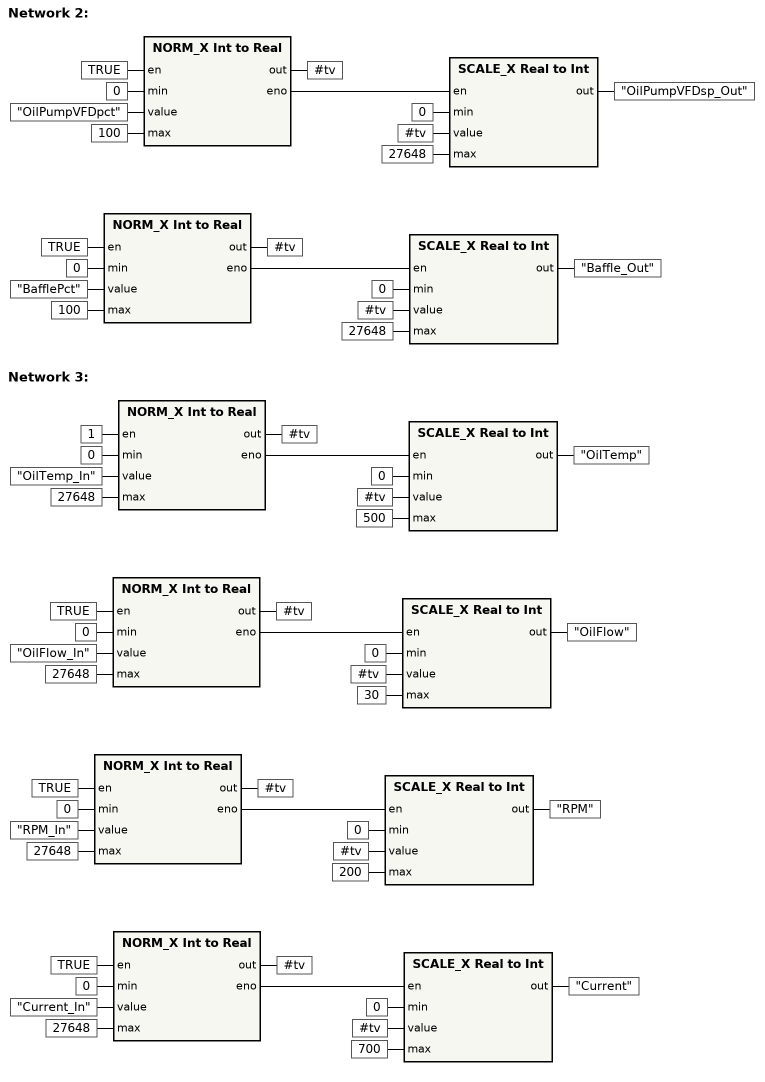
   IF TRUE THEN
       #tv := NORM_X(MIN := 0, VALUE := "OilPumpVFDpct", MAX := 100);
       "OilPumpVFDsp_Out" := SCALE_X(MIN := 0, VALUE := #tv, MAX := 27648);
       #tv := NORM_X(MIN := 0, VALUE := "BafflePct", MAX := 100);
       "Baffle_Out" := SCALE_X(MIN := 0, VALUE := #tv, MAX := 27648);
   END_IF;
END_REGION

REGION Network 3
   // Analog Inputs
   IF 1 THEN
       #tv := NORM_X(MIN := 0, VALUE := "OilTemp_In", MAX := 27648);
       "OilTemp" := SCALE_X(MIN := 0, VALUE := #tv, MAX := 500);
   END_IF;
   IF TRUE THEN
       #tv := NORM_X(MIN := 0, VALUE := "OilFlow_In", MAX := 27648);
       "OilFlow" := SCALE_X(MIN := 0, VALUE := #tv, MAX := 30);
       #tv := NORM_X(MIN := 0, VALUE := "RPM_In", MAX := 27648);
       "RPM" := SCALE_X(MIN := 0, VALUE := #tv, MAX := 200);
       #tv := NORM_X(MIN := 0, VALUE := "Current_In", MAX := 27648);
       "Current" := SCALE_X(MIN := 0, VALUE := #tv, MAX := 700);
   END_IF;
END_REGION
END_FUNCTION_BLOCK

FUNCTION_BLOCK "IO_STL"   // FB4, STL
{ S7_Optimized_Access := 'TRUE' }
VERSION : 0.1
BEGIN

REGION Network 1
   // Digital Outputs
         L     "OilPumpVFDhoa";
         L     0;
         ==I;
         JC    ResetOilPumpVFD;
         CLR;
         L     "OilPumpVFDhoa";
         L     1;
         ==I;
         JC    SetRunOilPumpVFD;
         CLR;
         L     "OilPumpVFDhoa";
         L     2;
         JC    AutoOilPumpVFD;


   AutoOilPumpVFD:A     "OilPumpVFD_Ctrl";
         JC    SetRunOilPumpVFD;
         JU    ResetOilPumpVFD;

   SetRunOilPumpVFD:S     "OilPumpVFDen_Out";
         JU    Brake;

   ResetOilPumpVFD:R     "OilPumpVFDen_Out";
         JU    Brake;


   Brake:L     "BrakeHoa";
         L     0;
         ==I;
         JC    ResetBrake;
         CLR;
         L     "BrakeHoa";
         L     1;
         ==I;
         JC    SetBrake;
         CLR;
         L     "BrakeHoa";
         L     2;
         ==I;
         JC    AutoBrake;

   AutoBrake:A     "Bracke_Ctrl";
         JC    SetBrake;
         JU    ResetBrake;

   ResetBrake:R     "Brake_Out";
         JU    AlarmHorn;
   SetBrake:S     "Brake_Out";
         JU    AlarmHorn;

   AlarmHorn:L     "AlarmHornHoa";
         L     0;
         ==I;
         JC    ResetAlarmHorn;
         CLR;
         L     "AlarmHornHoa";
         L     1;
         ==I;
         JC    SetAlarmHorn;
         CLR;
         L     "AlarmHornHoa";
         L     2;
         ==I;
         JC    AutoAlarmHorn;


   AutoAlarmHorn:A     "ALarmHorn_Ctrl";
         JC    SetAlarmHorn;
         JU    ResetAlarmHorn;


   SetAlarmHorn:S     "AlarmHorn_Out";
         JU    StationinterLock;

   ResetAlarmHorn:R     "AlarmHorn_Out";
         JU    StationinterLock;


   StationinterLock:L     "StationintHoa";
         L     0;
         ==I;
         JC    ResetStationinterLock;
         CLR;
         L     "StationintHoa";
         L     1;
         ==I;
         JC    SetStationinterLock;
         CLR;
         L     "StationintHoa";
         L     2;
         ==I;
         JC    AutoStationinterLock;
         JU    Baffle;



   AutoStationinterLock:A     "Stationint_Ctrl";
         JC    SetStationinterLock;
         JU    ResetStationinterLock;


   SetStationinterLock:S     "Stationinterlock_Out";
         JU    Baffle;
   ResetStationinterLock:R     "Stationinterlock_Out";
         JU    Baffle;



   Baffle:L     "BaffleHOA";
         L     0;
         ==I;
         JC    ResetStationinterLock;
         CLR;
         L     "StationintHoa";
         L     1;
         ==I;
         JC    SetStationinterLock;
         CLR;
         L     "StationintHoa";
         L     2;
         ==I;
         JC    AutoBaffle;
         JU    AnalogOutputs;



   AutoBaffle:A     "Baffle_Ctrl";
         JC    SetBaffle;
         JU    ResetBaffle;


   SetBaffle:S     "Baffle_En";
         JU    AnalogOutputs;
   ResetBaffle:R     "Baffle_En";
         JU    AnalogOutputs;

   // Analog Outputs

   AnalogOutputs:CALL  "SCP1"
         ( Input_Min    := 0,
           Input_Signal := "OilPumpVFDpct",
           Input_Max    := 100,
           Output_Min   := 0,
           Output_Max   := 27648,
           SV           := "OilPumpVFDsp_Out"
         );


         CALL  "SCP1"
         ( Input_Min    := 0,
           Input_Signal := "BafflePct",
           Input_Max    := 100,
           Output_Min   := 0,
           Output_Max   := 27648,
           SV           := "Baffle_Out"
         );



   // Analog Inputs

   AnalogInputs:CALL  "SCP1"
         ( Input_Min    := 0,
           Input_Signal := "OilTemp_In",
           Input_Max    := 27648,
           Output_Min   := 0,
           Output_Max   := 500,
           SV           := "OilTemp"
         );


         CALL  "SCP1"
         ( Input_Min    := 0,
           Input_Signal := "OilFlow_In",
           Input_Max    := 27648,
           Output_Min   := 0,
           Output_Max   := 30,
           SV           := "OilFlow"
         );



         CALL  "SCP1"
         ( Input_Min    := 0,
           Input_Signal := "RPM_In",
           Input_Max    := 27648,
           Output_Min   := 0,
           Output_Max   := 200,
           SV           := "RPM"
         );


         CALL  "SCP1"
         ( Input_Min    := 0,
           Input_Signal := "Current_In",
           Input_Max    := 27648,
           Output_Min   := 0,
           Output_Max   := 700,
           SV           := "Current"
         );
END_REGION
END_FUNCTION_BLOCK

FUNCTION_BLOCK "IO_SCL"   // FB5, SCL
{ S7_Optimized_Access := 'TRUE' }
VERSION : 0.1
BEGIN
   // Digital Outputs
   // Oil Pump VFD
   IF "OilPumpVFDhoa" = 0 THEN
       "OilPumpVFDen_Out" := 0;
   END_IF;

   IF "OilPumpVFDhoa" = 1 THEN
       "OilPumpVFDen_Out" := 1;
   END_IF;

   IF "OilPumpVFDhoa" = 2 AND "OilPumpVFD_Ctrl" THEN
       "OilPumpVFDen_Out" := 1;
   END_IF;

   IF "OilPumpVFDhoa" = 2 AND NOT "OilPumpVFD_Ctrl" THEN
       "OilPumpVFDsp_Out" := 0;
   END_IF;

   // Brake Output

   IF "BrakeHoa" = 0 OR   ("BrakeHoa" = 2 AND NOT "Bracke_Ctrl") THEN
       "Brake_Out" := 0;
   END_IF;

   IF "BrakeHoa" = 1 OR ("BrakeHoa" = 2 AND "Bracke_Ctrl") THEN
       "Brake_Out" := 1;
   END_IF;


   //Alarm Horn 

   IF "AlarmHornHoa" = 0 OR ("AlarmHornHoa" = 2 AND NOT "ALarmHorn_Ctrl") THEN
       "AlarmHorn_Out" := 0;
   END_IF;

   IF "AlarmHornHoa" = 1 OR ("AlarmHornHoa" = 2 AND "ALarmHorn_Ctrl") THEN
       "AlarmHorn_Out" := 1;
   END_IF;

   //Stationinterlock 

   IF "StationintHoa" = 0 OR ("StationintHoa" = 2 AND NOT "Stationint_Ctrl") THEN
       "Stationinterlock_Out" := 0;
   END_IF;

   IF "StationintHoa" = 1 OR ("StationintHoa" = 2 AND "Stationint_Ctrl") THEN
       "Stationinterlock_Out" := 1;
   END_IF;

   // Baffle 


   IF "BaffleHOA" = 0 OR ("BaffleHOA" = 2 AND NOT "Baffle_Ctrl") THEN
       "Baffle_En" := 0;
   END_IF;

   IF "BaffleHOA" = 1 OR ("BaffleHOA" = 2 AND "Baffle_Ctrl") THEN
       "Baffle_En" := 1;
   END_IF;


   // Analog Outputs
   "SCP1"(Input_Min:=0,
          Input_Signal:="OilPumpVFDpct",
          Input_Max:=100,
          Output_Min:=0,
          Output_Max:=27648,
          SV=>"OilPumpVFDsp_Out");

   "SCP1"(Input_Min:=0,
          Input_Signal:="BafflePct",
          Input_Max:=100,
          Output_Min:=0,
          Output_Max:=27648,
          SV=>"Baffle_Out");

   // Analog Inputs 

   "SCP1"(Input_Min:=0,
          Input_Signal:="OilTemp_In",
          Input_Max:=27648,
          Output_Min:=0,
          Output_Max:=500,
          SV=>"OilTemp");


   "SCP1"(Input_Min:=0,
          Input_Signal:="OilFlow_In",
          Input_Max:=27648,
          Output_Min:=0,
          Output_Max:=30,
          SV=>"OilFlow");


   "SCP1"(Input_Min:=0,
          Input_Signal:="RPM_In",
          Input_Max:=27648,
          Output_Min:=0,
          Output_Max:=200,
          SV=>"RPM");


   "SCP1"(Input_Min:=0,
          Input_Signal:="Current_In",
          Input_Max:=27648,
          Output_Min:=0,
          Output_Max:=700,
          SV=>"Current");
END_FUNCTION_BLOCK

FUNCTION_BLOCK "ALARMS_LAD"   // FB6, LAD
{ S7_Optimized_Access := 'TRUE' }
VERSION : 0.1
   VAR
      OS1 : Bool;
      OS2 : Bool;
      OS3 : Bool;
      OS5 : Bool;
      OS6 : Bool;
      OS4 : Bool;
      OS7 : Bool;
   END_VAR
   VAR_TEMP
      OLFD : Int;
      OLFAT : Bool;
      tv1 : Time;
      OCD : Int;
      tv2 : Time;
      OCAT : Bool;
      OTtd : Int;
      tv3 : Time;
      oiltempAT : Bool;
      RotTim : Int;
      tv4 : Time;
      OHFD : Int;
      RottAT : Bool;
      tv5 : Time;
      OHFAT : Bool;
      BFDT : Int;
      tv6 : Time;
      BFAT : Bool;
      ESAT : Bool;
   END_VAR
   VAR_TEMP   // added for the SCL form of the ladder/FBD networks
      _w1 : Bool;
      _w2 : Bool;
   END_VAR
BEGIN

REGION Network 1
   // Oil Low Flow Alarm
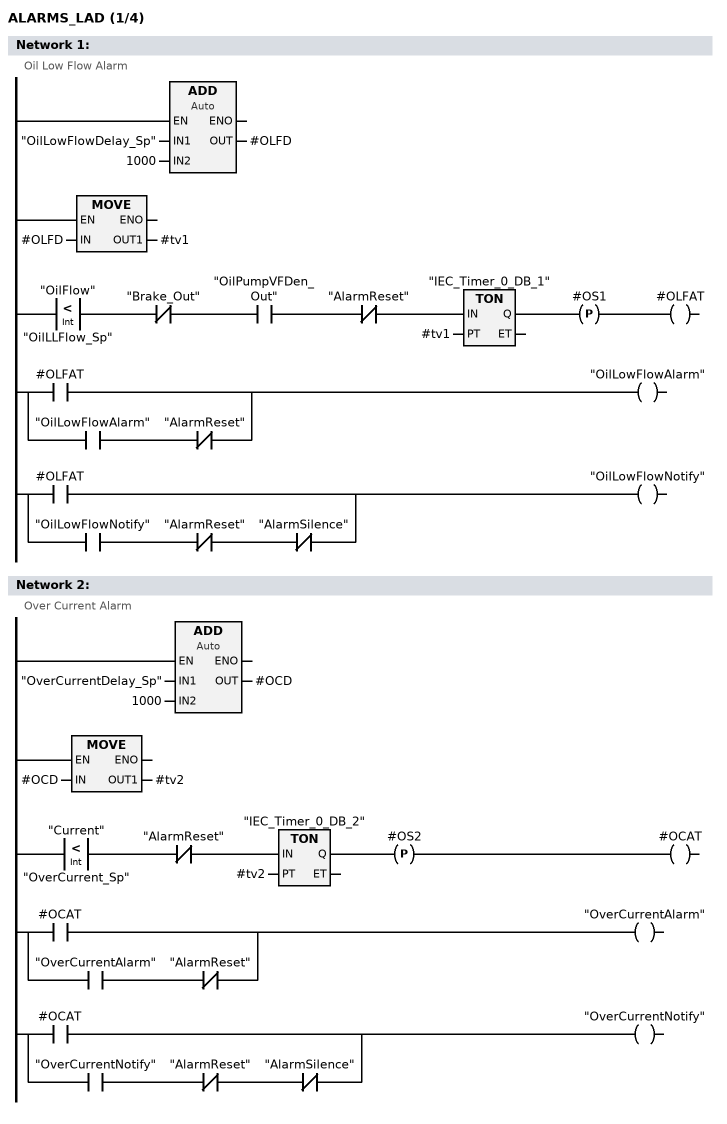
   #OLFD := "OilLowFlowDelay_Sp" + 1000;
   #tv1 := #OLFD;
   "IEC_Timer_0_DB_1".TON(IN := ("OilFlow" < "OilLLFlow_Sp") AND NOT "Brake_Out" AND "OilPumpVFDen_Out" AND NOT "AlarmReset",
                          PT := #tv1);
   #_w1 := "IEC_Timer_0_DB_1".Q AND NOT #OS1;   // rising edge
   #OS1 := "IEC_Timer_0_DB_1".Q;
   #OLFAT := #_w1;
   "OilLowFlowAlarm" := #OLFAT OR ("OilLowFlowAlarm" AND NOT "AlarmReset");
   "OilLowFlowNotify" := #OLFAT OR ("OilLowFlowNotify" AND NOT "AlarmReset" AND NOT "AlarmSilence");
END_REGION

REGION Network 2
   // Over Current Alarm
   #OCD := "OverCurrentDelay_Sp" + 1000;
   #tv2 := #OCD;
   "IEC_Timer_0_DB_2".TON(IN := ("Current" < "OverCurrent_Sp") AND NOT "AlarmReset", PT := #tv2);
   #_w1 := "IEC_Timer_0_DB_2".Q AND NOT #OS2;   // rising edge
   #OS2 := "IEC_Timer_0_DB_2".Q;
   #OCAT := #_w1;
   "OverCurrentAlarm" := #OCAT OR ("OverCurrentAlarm" AND NOT "AlarmReset");
   "OverCurrentNotify" := #OCAT OR ("OverCurrentNotify" AND NOT "AlarmReset" AND NOT "AlarmSilence");
END_REGION

REGION Network 3
   // High Oil Temp Alarm
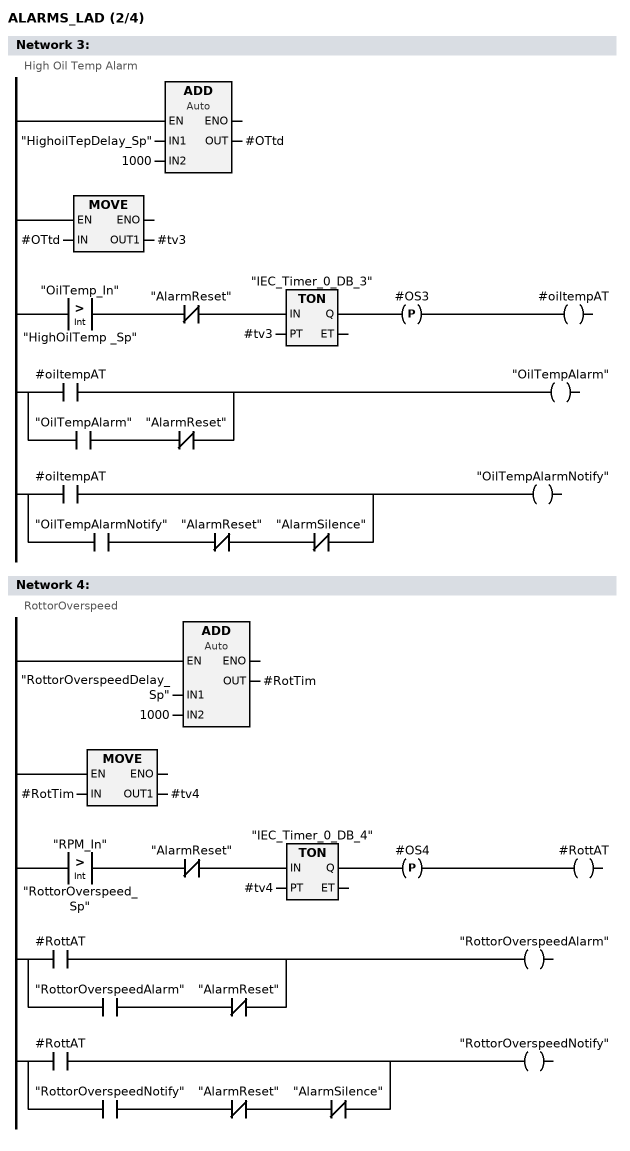
   #OTtd := "HighoilTepDelay_Sp" + 1000;
   #tv3 := #OTtd;
   "IEC_Timer_0_DB_3".TON(IN := ("OilTemp_In" > "HighOilTemp _Sp") AND NOT "AlarmReset", PT := #tv3);
   #_w1 := "IEC_Timer_0_DB_3".Q AND NOT #OS3;   // rising edge
   #OS3 := "IEC_Timer_0_DB_3".Q;
   #oiltempAT := #_w1;
   "OilTempAlarm" := #oiltempAT OR ("OilTempAlarm" AND NOT "AlarmReset");
   "OilTempAlarmNotify" := #oiltempAT OR ("OilTempAlarmNotify" AND NOT "AlarmReset" AND NOT "AlarmSilence");
END_REGION

REGION Network 4
   // RottorOverspeed
   #RotTim := "RottorOverspeedDelay_Sp" + 1000;
   #tv4 := #RotTim;
   "IEC_Timer_0_DB_4".TON(IN := ("RPM_In" > "RottorOverspeed_Sp") AND NOT "AlarmReset", PT := #tv4);
   #_w1 := "IEC_Timer_0_DB_4".Q AND NOT #OS4;   // rising edge
   #OS4 := "IEC_Timer_0_DB_4".Q;
   #RottAT := #_w1;
   "RottorOverspeedAlarm" := #RottAT OR ("RottorOverspeedAlarm" AND NOT "AlarmReset");
   "RottorOverspeedNotify" := #RottAT OR ("RottorOverspeedNotify" AND NOT "AlarmReset" AND NOT "AlarmSilence");
END_REGION

REGION Network 5
   // Oil High Flow Alarm
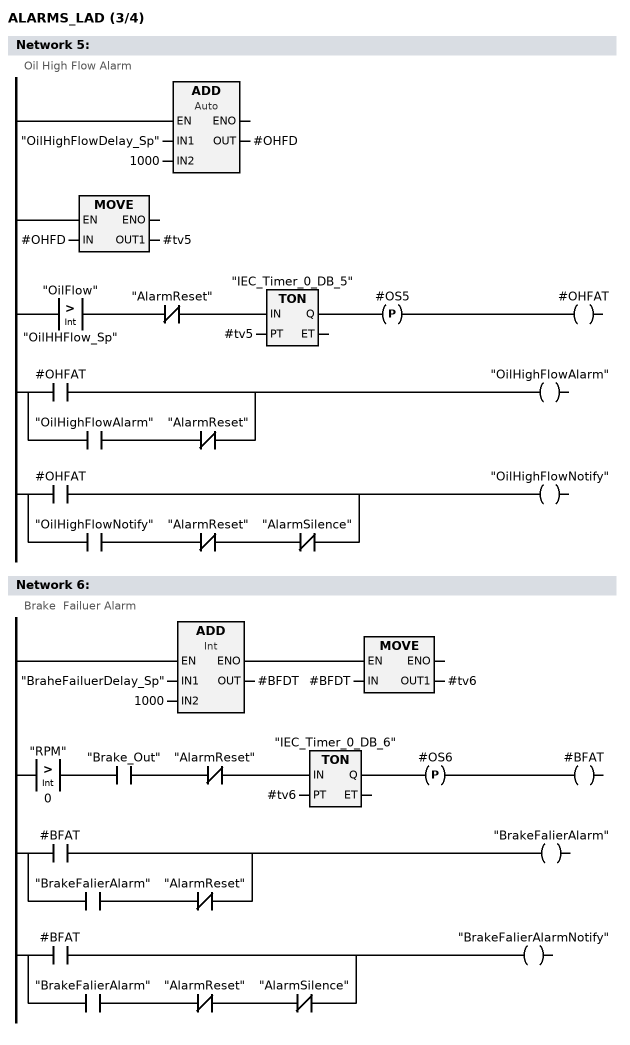
   #OHFD := "OilHighFlowDelay_Sp" + 1000;
   #tv5 := #OHFD;
   "IEC_Timer_0_DB_5".TON(IN := ("OilFlow" > "OilHHFlow_Sp") AND NOT "AlarmReset", PT := #tv5);
   #_w1 := "IEC_Timer_0_DB_5".Q AND NOT #OS5;   // rising edge
   #OS5 := "IEC_Timer_0_DB_5".Q;
   #OHFAT := #_w1;
   "OilHighFlowAlarm" := #OHFAT OR ("OilHighFlowAlarm" AND NOT "AlarmReset");
   "OilHighFlowNotify" := #OHFAT OR ("OilHighFlowNotify" AND NOT "AlarmReset" AND NOT "AlarmSilence");
END_REGION

REGION Network 6
   // Brake  Failuer Alarm
   #BFDT := "BraheFailuerDelay_Sp" + 1000;
   #tv6 := #BFDT;
   "IEC_Timer_0_DB_6".TON(IN := ("RPM" > 0) AND "Brake_Out" AND NOT "AlarmReset", PT := #tv6);
   #_w1 := "IEC_Timer_0_DB_6".Q AND NOT #OS6;   // rising edge
   #OS6 := "IEC_Timer_0_DB_6".Q;
   #BFAT := #_w1;
   "BrakeFalierAlarm" := #BFAT OR ("BrakeFalierAlarm" AND NOT "AlarmReset");
   "BrakeFalierAlarmNotify" := #BFAT OR ("BrakeFalierAlarm" AND NOT "AlarmReset" AND NOT "AlarmSilence");
END_REGION

REGION Network 7
   // EStop
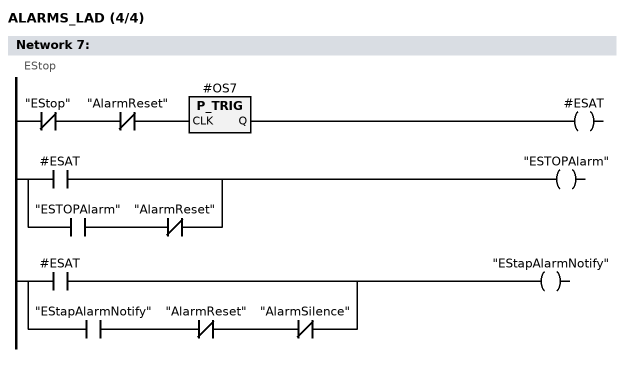
   RUNG wire#powerrail
      I_Contact( "EStop" )
      I_Contact( "AlarmReset" )
      P_Trig( #OS7 )
      Coil( #ESAT )
   END_RUNG
   RUNG wire#powerrail
      Contact( #ESAT )
      wire#w1
      Coil( "ESTOPAlarm" )
   END_RUNG
   RUNG wire#powerrail
      Contact( "ESTOPAlarm" )
      I_Contact( "AlarmReset" )
   END_RUNG wire#w1
   RUNG wire#powerrail
      Contact( #ESAT )
      wire#w2
      Coil( "EStapAlarmNotify" )
   END_RUNG
   RUNG wire#powerrail
      Contact( "EStapAlarmNotify" )
      I_Contact( "AlarmReset" )
      I_Contact( "AlarmSilence" )
   END_RUNG wire#w2
   // the same network as SCL:
   #_w1 := NOT "EStop" AND NOT "AlarmReset";
   #_w2 := #_w1 AND NOT #OS7;   // rising edge
   #OS7 := #_w1;
   #ESAT := #_w2;
   "ESTOPAlarm" := #ESAT OR ("ESTOPAlarm" AND NOT "AlarmReset");
   "EStapAlarmNotify" := #ESAT OR ("EStapAlarmNotify" AND NOT "AlarmReset" AND NOT "AlarmSilence");
END_REGION
END_FUNCTION_BLOCK

FUNCTION_BLOCK "SCP"   // FB7, FBD
{ S7_Optimized_Access := 'TRUE' }
VERSION : 0.1
   VAR_INPUT
      Input_Min : Int;
      Input_Max : Int;
      Input_Signal : Int;
      Output_Min : Int;
      Output_Max : Int;
   END_VAR
   VAR_OUTPUT
      SV : Int;
   END_VAR
   VAR_TEMP
      tv : Real;
   END_VAR
BEGIN

REGION Network 1
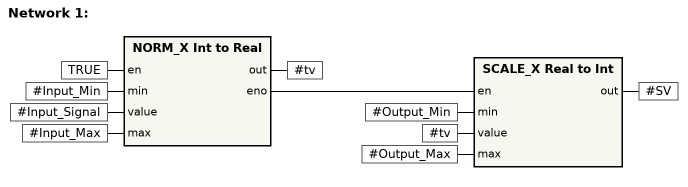
   IF TRUE THEN
       #tv := NORM_X(MIN := #Input_Min, VALUE := #Input_Signal, MAX := #Input_Max);
       #SV := SCALE_X(MIN := #Output_Min, VALUE := #tv, MAX := #Output_Max);
   END_IF;
END_REGION
END_FUNCTION_BLOCK

FUNCTION_BLOCK "HOA_LAD"   // FB8, LAD
{ S7_Optimized_Access := 'TRUE' }
VERSION : 0.1
   VAR
      OS1 : Bool;
      OS2 : Bool;
      OS3 : Bool;
      OS4 : Bool;
      OS5 : Bool;
      OS6 : Bool;
      OS7 : Bool;
      OS8 : Bool;
      OS9 : Bool;
      OS10 : Bool;
      OS11 : Bool;
      OS12 : Bool;
   END_VAR
   VAR_TEMP   // added for the SCL form of the ladder/FBD networks
      _w1 : Bool;
      _w2 : Bool;
      _w3 : Bool;
   END_VAR
BEGIN

REGION Network 1
   // Brake
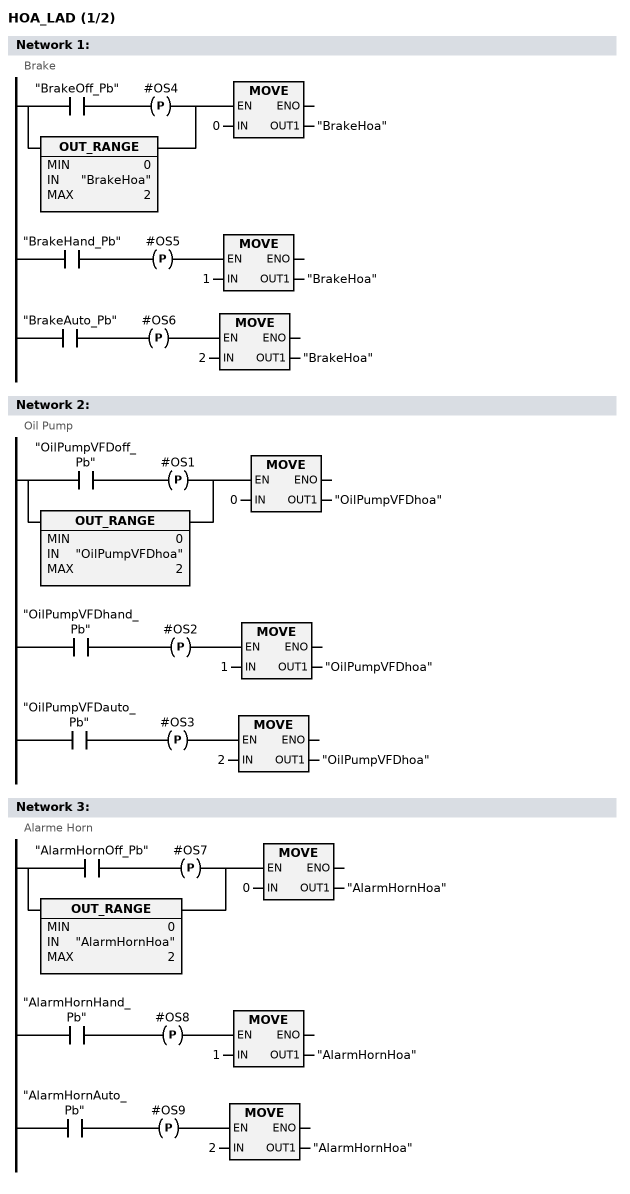
   #_w1 := "BrakeOff_Pb" AND NOT #OS4;   // rising edge
   #OS4 := "BrakeOff_Pb";
   IF #_w1 OR ("BrakeHoa" < 0) OR ("BrakeHoa" > 2) THEN "BrakeHoa" := 0; END_IF;
   #_w2 := "BrakeHand_Pb" AND NOT #OS5;   // rising edge
   #OS5 := "BrakeHand_Pb";
   IF #_w2 THEN "BrakeHoa" := 1; END_IF;
   #_w3 := "BrakeAuto_Pb" AND NOT #OS6;   // rising edge
   #OS6 := "BrakeAuto_Pb";
   IF #_w3 THEN "BrakeHoa" := 2; END_IF;
END_REGION

REGION Network 2
   // Oil Pump
   #_w1 := "OilPumpVFDoff_Pb" AND NOT #OS1;   // rising edge
   #OS1 := "OilPumpVFDoff_Pb";
   IF #_w1 OR ("OilPumpVFDhoa" < 0) OR ("OilPumpVFDhoa" > 2) THEN "OilPumpVFDhoa" := 0; END_IF;
   #_w2 := "OilPumpVFDhand_Pb" AND NOT #OS2;   // rising edge
   #OS2 := "OilPumpVFDhand_Pb";
   IF #_w2 THEN "OilPumpVFDhoa" := 1; END_IF;
   #_w3 := "OilPumpVFDauto_Pb" AND NOT #OS3;   // rising edge
   #OS3 := "OilPumpVFDauto_Pb";
   IF #_w3 THEN "OilPumpVFDhoa" := 2; END_IF;
END_REGION

REGION Network 3
   // Alarme Horn
   #_w1 := "AlarmHornOff_Pb" AND NOT #OS7;   // rising edge
   #OS7 := "AlarmHornOff_Pb";
   IF #_w1 OR ("AlarmHornHoa" < 0) OR ("AlarmHornHoa" > 2) THEN "AlarmHornHoa" := 0; END_IF;
   #_w2 := "AlarmHornHand_Pb" AND NOT #OS8;   // rising edge
   #OS8 := "AlarmHornHand_Pb";
   IF #_w2 THEN "AlarmHornHoa" := 1; END_IF;
   #_w3 := "AlarmHornAuto_Pb" AND NOT #OS9;   // rising edge
   #OS9 := "AlarmHornAuto_Pb";
   IF #_w3 THEN "AlarmHornHoa" := 2; END_IF;
END_REGION

REGION Network 4
   // Stationinterlock
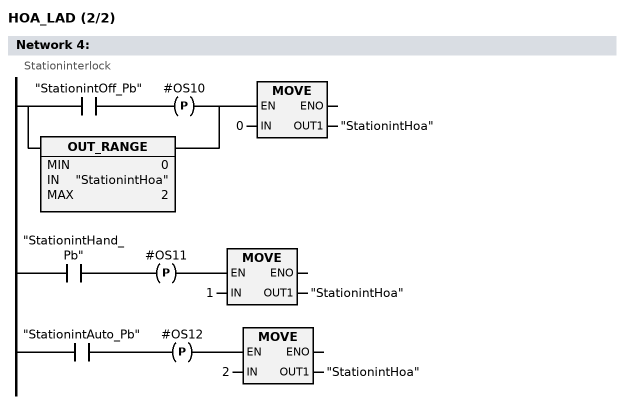
   #_w1 := "StationintOff_Pb" AND NOT #OS10;   // rising edge
   #OS10 := "StationintOff_Pb";
   IF #_w1 OR ("StationintHoa" < 0) OR ("StationintHoa" > 2) THEN "StationintHoa" := 0; END_IF;
   #_w2 := "StationintHand_Pb" AND NOT #OS11;   // rising edge
   #OS11 := "StationintHand_Pb";
   IF #_w2 THEN "StationintHoa" := 1; END_IF;
   #_w3 := "StationintAuto_Pb" AND NOT #OS12;   // rising edge
   #OS12 := "StationintAuto_Pb";
   IF #_w3 THEN "StationintHoa" := 2; END_IF;
END_REGION
END_FUNCTION_BLOCK

FUNCTION_BLOCK "HOA_FBD"   // FB9, FBD
{ S7_Optimized_Access := 'TRUE' }
VERSION : 0.1
   VAR
      OS1 : Bool;
      OS2 : Bool;
      OS3 : Bool;
      OS4 : Bool;
      OS5 : Bool;
      OS6 : Bool;
      OS7 : Bool;
      OS8 : Bool;
      OS9 : Bool;
      OS10 : Bool;
      OS11 : Bool;
      OS12 : Bool;
   END_VAR
   VAR_TEMP   // added for the SCL form of the ladder/FBD networks
      _w1 : Bool;
      _w2 : Bool;
      _w3 : Bool;
   END_VAR
BEGIN

REGION Network 1
   // Oil Pump
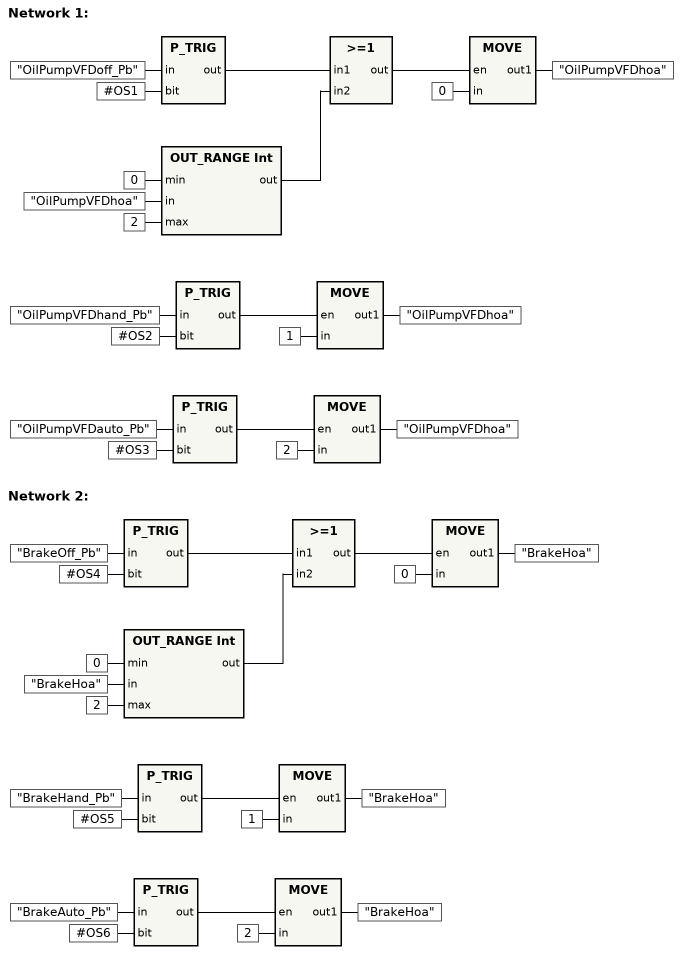
   #_w1 := "OilPumpVFDoff_Pb" AND NOT #OS1;   // rising edge
   #OS1 := "OilPumpVFDoff_Pb";
   IF #_w1 OR ("OilPumpVFDhoa" < 0) OR ("OilPumpVFDhoa" > 2) THEN "OilPumpVFDhoa" := 0; END_IF;
   #_w2 := "OilPumpVFDhand_Pb" AND NOT #OS2;   // rising edge
   #OS2 := "OilPumpVFDhand_Pb";
   IF #_w2 THEN "OilPumpVFDhoa" := 1; END_IF;
   #_w3 := "OilPumpVFDauto_Pb" AND NOT #OS3;   // rising edge
   #OS3 := "OilPumpVFDauto_Pb";
   IF #_w3 THEN "OilPumpVFDhoa" := 2; END_IF;
END_REGION

REGION Network 2
   // Brake
   #_w1 := "BrakeOff_Pb" AND NOT #OS4;   // rising edge
   #OS4 := "BrakeOff_Pb";
   IF #_w1 OR ("BrakeHoa" < 0) OR ("BrakeHoa" > 2) THEN "BrakeHoa" := 0; END_IF;
   #_w2 := "BrakeHand_Pb" AND NOT #OS5;   // rising edge
   #OS5 := "BrakeHand_Pb";
   IF #_w2 THEN "BrakeHoa" := 1; END_IF;
   #_w3 := "BrakeAuto_Pb" AND NOT #OS6;   // rising edge
   #OS6 := "BrakeAuto_Pb";
   IF #_w3 THEN "BrakeHoa" := 2; END_IF;
END_REGION

REGION Network 3
   // Alarme Horn
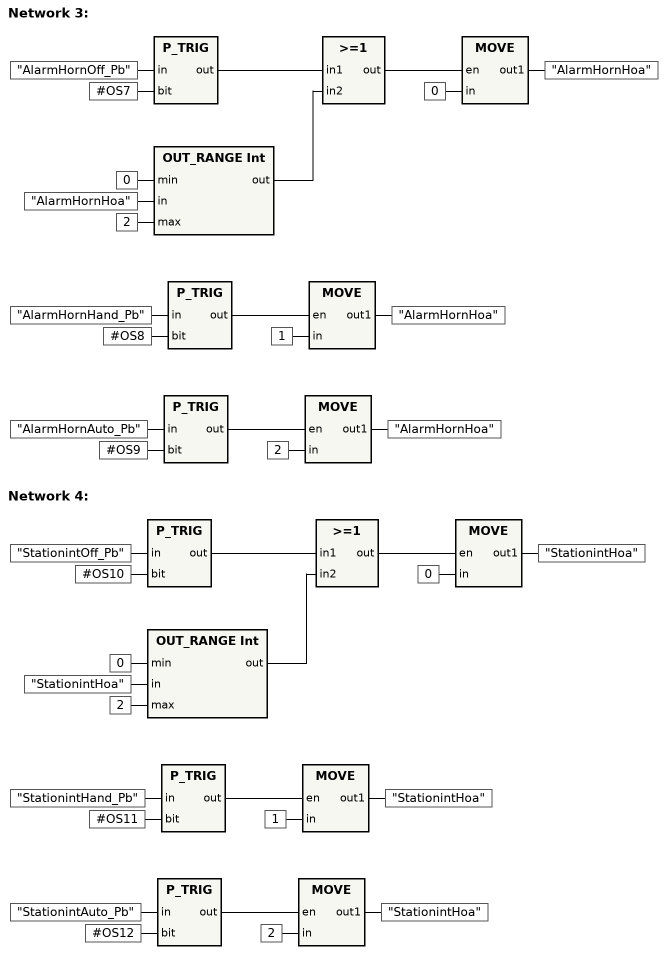
   #_w1 := "AlarmHornOff_Pb" AND NOT #OS7;   // rising edge
   #OS7 := "AlarmHornOff_Pb";
   IF #_w1 OR ("AlarmHornHoa" < 0) OR ("AlarmHornHoa" > 2) THEN "AlarmHornHoa" := 0; END_IF;
   #_w2 := "AlarmHornHand_Pb" AND NOT #OS8;   // rising edge
   #OS8 := "AlarmHornHand_Pb";
   IF #_w2 THEN "AlarmHornHoa" := 1; END_IF;
   #_w3 := "AlarmHornAuto_Pb" AND NOT #OS9;   // rising edge
   #OS9 := "AlarmHornAuto_Pb";
   IF #_w3 THEN "AlarmHornHoa" := 2; END_IF;
END_REGION

REGION Network 4
   // Stationinterlock
   #_w1 := "StationintOff_Pb" AND NOT #OS10;   // rising edge
   #OS10 := "StationintOff_Pb";
   IF #_w1 OR ("StationintHoa" < 0) OR ("StationintHoa" > 2) THEN "StationintHoa" := 0; END_IF;
   #_w2 := "StationintHand_Pb" AND NOT #OS11;   // rising edge
   #OS11 := "StationintHand_Pb";
   IF #_w2 THEN "StationintHoa" := 1; END_IF;
   #_w3 := "StationintAuto_Pb" AND NOT #OS12;   // rising edge
   #OS12 := "StationintAuto_Pb";
   IF #_w3 THEN "StationintHoa" := 2; END_IF;
END_REGION
END_FUNCTION_BLOCK

FUNCTION_BLOCK "HOA_STL"   // FB10, STL
{ S7_Optimized_Access := 'TRUE' }
VERSION : 0.1
   VAR
      OS1 : Bool;
      OS2 : Bool;
      OS3 : Bool;
      OS4 : Bool;
      OS5 : Bool;
      OS6 : Bool;
      OS7 : Bool;
      OS8 : Bool;
      OS9 : Bool;
      OS10 : Bool;
      OS11 : Bool;
      OS12 : Bool;
   END_VAR
BEGIN

REGION Network 1
         L     "OilPumpVFDhoa";
         L     0;
         <I;
         JC    SetOilPumpVFDHoaZero;
         CLR;
         L     "OilPumpVFDhoa";
         L     2;
         >I;
         JC    SetOilPumpVFDHoaZero;
         CLR;
         A     "OilPumpVFDoff_Pb";
         FP    #OS1;
         JC    SetOilPumpVFDHoaZero;
         CLR;
         A     "OilPumpVFDhand_Pb";
         FP    #OS2;
         JC    SetOilPumpVFDHoaOne;
         CLR;
         A     "OilPumpVFDauto_Pb";
         FP    #OS3;
         JC    SetOilPumpVFDHoaTwo;
         JU    Brake;


   SetOilPumpVFDHoaZero:L     0;
         T     "OilPumpVFDhoa";
         JU    Brake;
   SetOilPumpVFDHoaOne:L     1;
         T     "OilPumpVFDhoa";
         JU    Brake;
   SetOilPumpVFDHoaTwo:L     2;
         T     "OilPumpVFDhoa";
         JU    Brake;


   Brake:L     "BrakeHoa";
         L     0;
         <I;
         JC    SetBrakeZero;
         CLR;
         L     "BrakeHoa";
         L     2;
         >I;
         JC    SetBrakeZero;
         CLR;
         A     "BrakeOff_Pb";
         FP    #OS4;
         JC    SetBrakeZero;
         CLR;
         A     "BrakeHand_Pb";
         FP    #OS5;
         JC    SetBrakeOne;
         CLR;
         A     "BrakeAuto_Pb";
         FP    #OS6;
         JC    SetBrakeTwo;
         JU    AlarmHorn;


   SetBrakeZero:L     0;
         T     "BrakeHoa";
         JU    AlarmHorn;
   SetBrakeOne:L     1;
         T     "BrakeHoa";
         JU    AlarmHorn;
   SetBrakeTwo:L     2;
         T     "BrakeHoa";
         JU    AlarmHorn;

   AlarmHorn:L     "AlarmHornHoa";
         L     0;
         <I;
         JC    SetAlarmHornZero;
         CLR;
         L     "AlarmHornHoa";
         L     2;
         >I;
         JC    SetAlarmHornZero;
         CLR;
         A     "AlarmHornOff_Pb";
         FP    #OS7;
         JC    SetAlarmHornZero;
         CLR;
         A     "AlarmHornHand_Pb";
         FP    #OS8;
         JC    SetAlarnHornOne;
         CLR;
         A     "AlarmHornAuto_Pb";
         FP    #OS9;
         JC    SetAlarmHornTwe;
         JU    StationInterlock;






   SetAlarmHornZero:L     0;
         L     "AlarmHornHoa";
         JU    StationInterlock;
   SetAlarnHornOne:L     1;
         L     "AlarmHornHoa";
         JU    StationInterlock;
   SetAlarmHornTwe:L     2;
         L     "AlarmHornHoa";
         JU    StationInterlock;


   StationInterlock:L     "StationintHoa";
         L     0;
         <I;
         JC    SetStationinterZero;
         CLR;
         L     "StationintHoa";
         L     2;
         >I;
         JC    SetStationinterZero;
         CLR;
         A     "StationintOff_Pb";
         FP    #OS10;
         JC    SetStationinterZero;
         CLR;
         A     "StationintHand_Pb";
         FP    #OS11;
         JC    SetStationinterOne;
         CLR;
         A     "StationintAuto_Pb";
         FP    #OS12;
         JC    SetStationinterTwe;
         JU    EndOfLine;



   SetStationinterZero:L     0;
         L     "StationintHoa";
         BE;
   SetStationinterOne:L     1;
         L     "StationintHoa";
         BE;
   SetStationinterTwe:L     2;
         L     "StationintHoa";
         BE;

   EndOfLine:BE;
END_REGION
END_FUNCTION_BLOCK

FUNCTION_BLOCK "HOA_SCL"   // FB11, SCL
{ S7_Optimized_Access := 'TRUE' }
VERSION : 0.1
BEGIN
   // Oil Pump VFD HOA Controls 

   IF "OilPumpVFDhoa" < 0 OR "OilPumpVFDhoa" > 2  THEN
       "OilPumpVFDhoa" := 0;
   END_IF;


   IF "OilPumpVFDoff_Pb" AND "OilPumpVFDhoa" <> 0 THEN
       "OilPumpVFDhoa" := 0;
   END_IF;

   IF "OilPumpVFDhand_Pb"  AND "OilPumpVFDhoa" <> 1 THEN
       "OilPumpVFDhoa" := 1;
   END_IF;

   IF "OilPumpVFDauto_Pb"  AND "OilPumpVFDhoa" <> 2 THEN
       "OilPumpVFDhoa" := 2;
   END_IF;

   // Brakes HOA Controls 

   IF "BrakeHoa" < 0 OR "BrakeHoa" > 2 THEN
       "BrakeHoa" := 0;
   END_IF;

   IF "BrakeOff_Pb" AND "BrakeHoa" <> 0 THEN
       "BrakeHoa" := 0;
   END_IF;

   IF "BrakeHand_Pb" AND "BrakeHoa" <> 1 THEN
       "BrakeHoa" := 1;
   END_IF;

   IF "BrakeAuto_Pb" AND "BrakeHoa" <> 2 THEN
       "BrakeHoa" := 2;
   END_IF;

   //AlarmHorn HOA Controls 

   IF "AlarmHornHoa" < 0 OR "AlarmHornHoa" > 2 THEN
       "AlarmHornHoa" := 0;
   END_IF;

   IF "AlarmHornOff_Pb" AND "AlarmHornHoa" <> 0 THEN
       "AlarmHornHoa" := 0;
   END_IF;

   IF "AlarmHornHand_Pb" AND "AlarmHornHoa" <> 1 THEN
       "AlarmHornHoa" := 1;
   END_IF;

   IF "AlarmHornAuto_Pb" AND "AlarmHornHoa" <> 2 THEN
       "AlarmHornHoa" := 2;
   END_IF;

   //  StationinterLock HOA Controls 

   IF "StationintHoa" < 0 OR "StationintHoa" > 2 THEN
       "StationintHoa" := 0;
   END_IF;

   IF "StationintOff_Pb" AND "StationintHoa" <> 0 THEN
       "StationintHoa" := 0;
   END_IF;

   IF "StationintHand_Pb" AND "StationintHoa" <> 1 THEN
       "StationintHoa" := 1;
   END_IF;

   IF "StationintAuto_Pb" AND "StationintHoa" <> 2 THEN
       "StationintHoa" := 2;
   END_IF;
END_FUNCTION_BLOCK

FUNCTION_BLOCK "ALARMS_FBD"   // FB12, FBD
{ S7_Optimized_Access := 'TRUE' }
VERSION : 0.1
   VAR
      OS1 : Bool;
      OS2 : Bool;
      OS3 : Bool;
      OS4 : Bool;
      OS5 : Bool;
      OS6 : Bool;
      OS7 : Bool;
   END_VAR
   VAR_TEMP
      ti1 : Int;
      tt1 : Time;
      tt2 : Time;
      ti2 : Int;
      ti3 : Int;
      tt3 : Time;
      tt4 : Time;
      ti4 : Int;
      tt5 : Time;
      ti5 : Int;
      tt6 : Time;
      ti6 : Int;
   END_VAR
   VAR_TEMP   // added for the SCL form of the ladder/FBD networks
      _w1 : Bool;
   END_VAR
BEGIN

REGION Network 1
   // Oil Low Flow Alarm
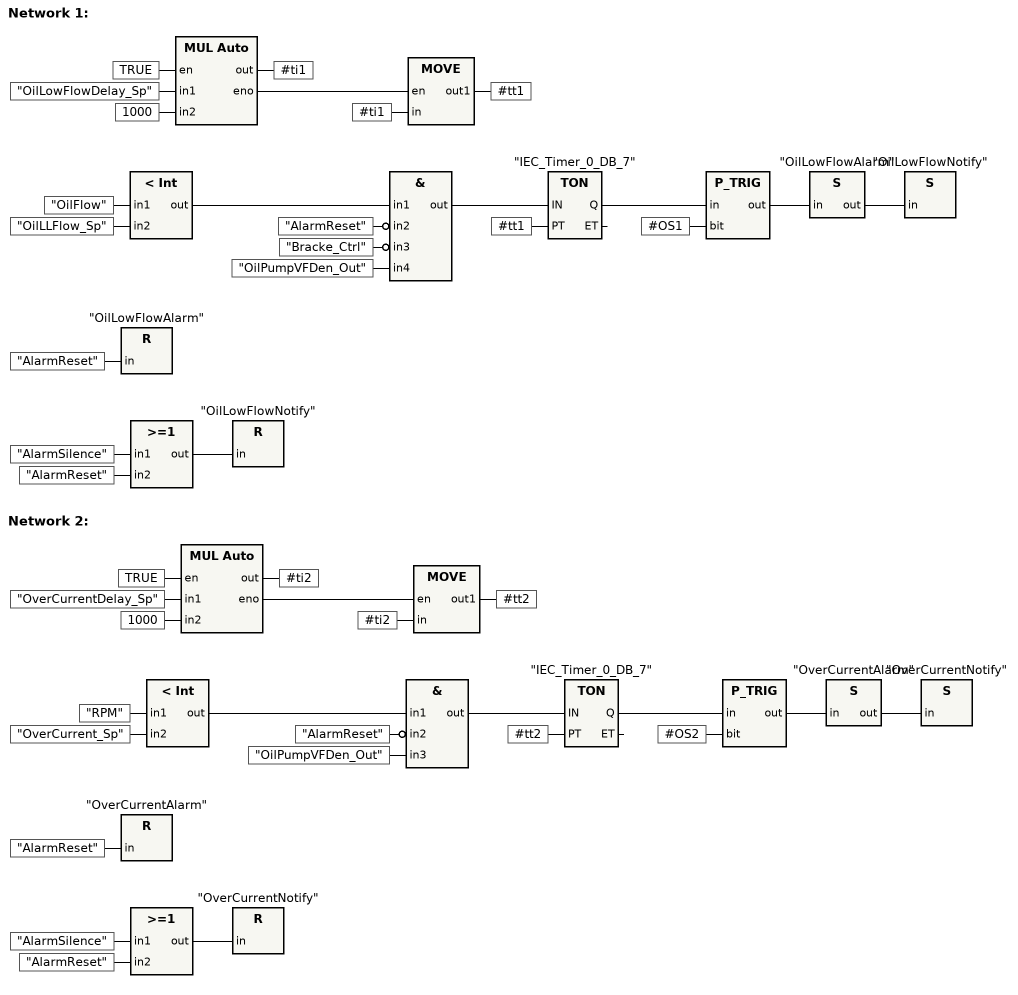
   IF TRUE THEN
       #ti1 := "OilLowFlowDelay_Sp" * 1000;
       #tt1 := #ti1;
   END_IF;
   "IEC_Timer_0_DB_7".TON(IN := ("OilFlow" < "OilLLFlow_Sp") AND NOT "AlarmReset" AND NOT "Bracke_Ctrl" AND "OilPumpVFDen_Out",
                          PT := #tt1);
   #_w1 := "IEC_Timer_0_DB_7".Q AND NOT #OS1;   // rising edge
   #OS1 := "IEC_Timer_0_DB_7".Q;
   IF #_w1 THEN
       "OilLowFlowAlarm" := TRUE;
       "OilLowFlowNotify" := TRUE;
   END_IF;
   IF "AlarmReset" THEN "OilLowFlowAlarm" := FALSE; END_IF;
   IF "AlarmSilence" OR "AlarmReset" THEN "OilLowFlowNotify" := FALSE; END_IF;
END_REGION

REGION Network 2
   // Over Current
   IF TRUE THEN
       #ti2 := "OverCurrentDelay_Sp" * 1000;
       #tt2 := #ti2;
   END_IF;
   "IEC_Timer_0_DB_7".TON(IN := ("RPM" < "OverCurrent_Sp") AND NOT "AlarmReset" AND "OilPumpVFDen_Out",
                          PT := #tt2);
   #_w1 := "IEC_Timer_0_DB_7".Q AND NOT #OS2;   // rising edge
   #OS2 := "IEC_Timer_0_DB_7".Q;
   IF #_w1 THEN
       "OverCurrentAlarm" := TRUE;
       "OverCurrentNotify" := TRUE;
   END_IF;
   IF "AlarmReset" THEN "OverCurrentAlarm" := FALSE; END_IF;
   IF "AlarmSilence" OR "AlarmReset" THEN "OverCurrentNotify" := FALSE; END_IF;
END_REGION

REGION Network 3
   // High Oil Temp Alarm
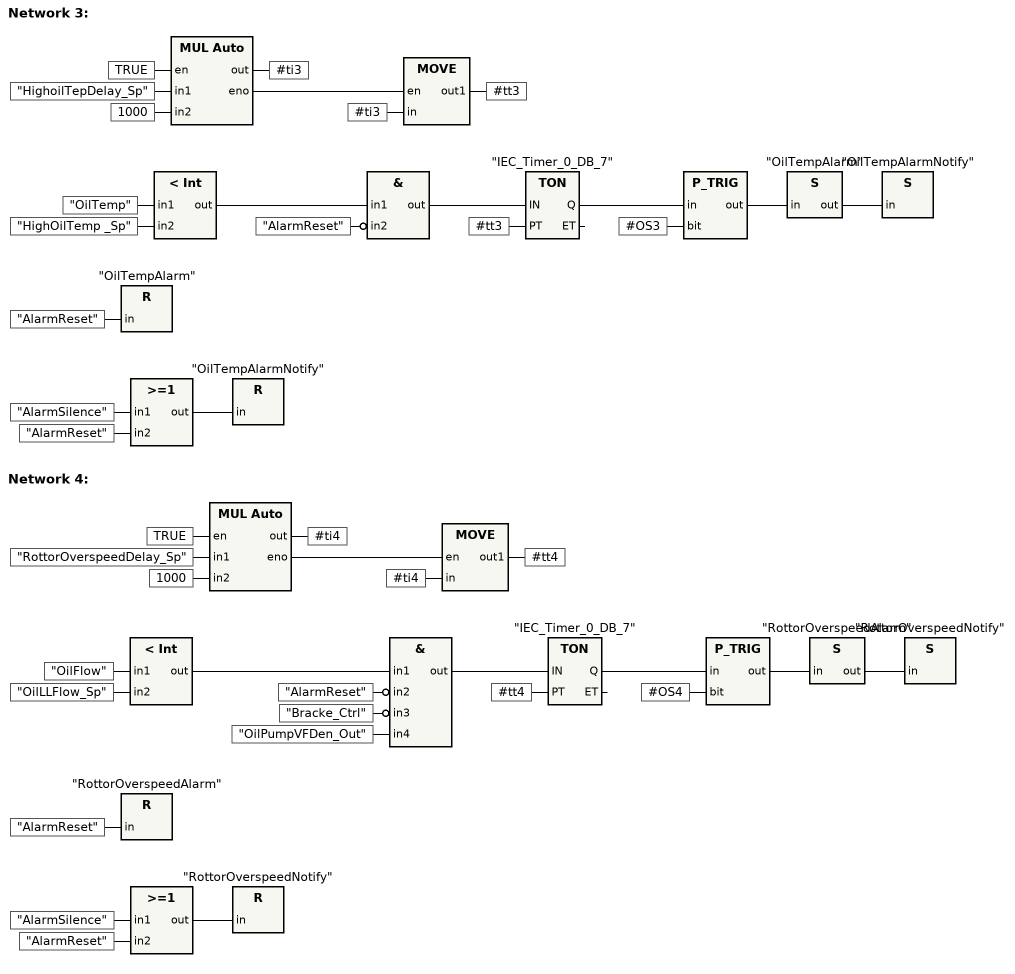
   IF TRUE THEN
       #ti3 := "HighoilTepDelay_Sp" * 1000;
       #tt3 := #ti3;
   END_IF;
   "IEC_Timer_0_DB_7".TON(IN := ("OilTemp" < "HighOilTemp _Sp") AND NOT "AlarmReset", PT := #tt3);
   #_w1 := "IEC_Timer_0_DB_7".Q AND NOT #OS3;   // rising edge
   #OS3 := "IEC_Timer_0_DB_7".Q;
   IF #_w1 THEN
       "OilTempAlarm" := TRUE;
       "OilTempAlarmNotify" := TRUE;
   END_IF;
   IF "AlarmReset" THEN "OilTempAlarm" := FALSE; END_IF;
   IF "AlarmSilence" OR "AlarmReset" THEN "OilTempAlarmNotify" := FALSE; END_IF;
END_REGION

REGION Network 4
   // RottorOverspeed
   IF TRUE THEN
       #ti4 := "RottorOverspeedDelay_Sp" * 1000;
       #tt4 := #ti4;
   END_IF;
   "IEC_Timer_0_DB_7".TON(IN := ("OilFlow" < "OilLLFlow_Sp") AND NOT "AlarmReset" AND NOT "Bracke_Ctrl" AND "OilPumpVFDen_Out",
                          PT := #tt4);
   #_w1 := "IEC_Timer_0_DB_7".Q AND NOT #OS4;   // rising edge
   #OS4 := "IEC_Timer_0_DB_7".Q;
   IF #_w1 THEN
       "RottorOverspeedAlarm" := TRUE;
       "RottorOverspeedNotify" := TRUE;
   END_IF;
   IF "AlarmReset" THEN "RottorOverspeedAlarm" := FALSE; END_IF;
   IF "AlarmSilence" OR "AlarmReset" THEN "RottorOverspeedNotify" := FALSE; END_IF;
END_REGION

REGION Network 5
   // Oil High Flow Alarm
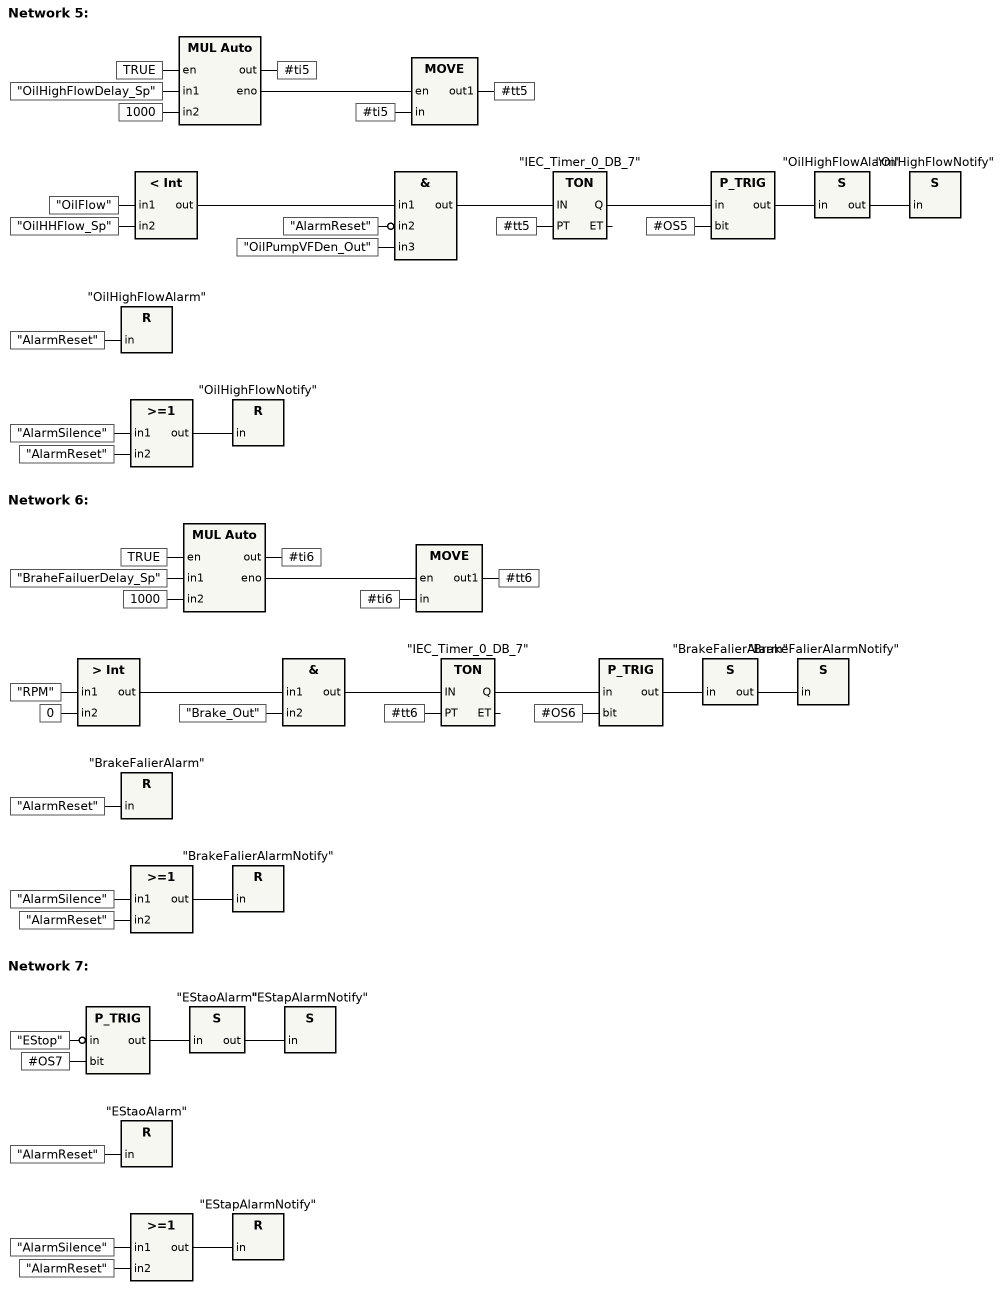
   IF TRUE THEN
       #ti5 := "OilHighFlowDelay_Sp" * 1000;
       #tt5 := #ti5;
   END_IF;
   "IEC_Timer_0_DB_7".TON(IN := ("OilFlow" < "OilHHFlow_Sp") AND NOT "AlarmReset" AND "OilPumpVFDen_Out",
                          PT := #tt5);
   #_w1 := "IEC_Timer_0_DB_7".Q AND NOT #OS5;   // rising edge
   #OS5 := "IEC_Timer_0_DB_7".Q;
   IF #_w1 THEN
       "OilHighFlowAlarm" := TRUE;
       "OilHighFlowNotify" := TRUE;
   END_IF;
   IF "AlarmReset" THEN "OilHighFlowAlarm" := FALSE; END_IF;
   IF "AlarmSilence" OR "AlarmReset" THEN "OilHighFlowNotify" := FALSE; END_IF;
END_REGION

REGION Network 6
   // Brake  Failuer Alarm
   IF TRUE THEN
       #ti6 := "BraheFailuerDelay_Sp" * 1000;
       #tt6 := #ti6;
   END_IF;
   "IEC_Timer_0_DB_7".TON(IN := ("RPM" > 0) AND "Brake_Out", PT := #tt6);
   #_w1 := "IEC_Timer_0_DB_7".Q AND NOT #OS6;   // rising edge
   #OS6 := "IEC_Timer_0_DB_7".Q;
   IF #_w1 THEN
       "BrakeFalierAlarm" := TRUE;
       "BrakeFalierAlarmNotify" := TRUE;
   END_IF;
   IF "AlarmReset" THEN "BrakeFalierAlarm" := FALSE; END_IF;
   IF "AlarmSilence" OR "AlarmReset" THEN "BrakeFalierAlarmNotify" := FALSE; END_IF;
END_REGION

REGION Network 7
   // EStop
   #_w1 := NOT "EStop" AND NOT #OS7;   // rising edge
   #OS7 := NOT "EStop";
   IF #_w1 THEN
       "EStaoAlarm" := TRUE;
       "EStapAlarmNotify" := TRUE;
   END_IF;
   IF "AlarmReset" THEN "EStaoAlarm" := FALSE; END_IF;
   IF "AlarmSilence" OR "AlarmReset" THEN "EStapAlarmNotify" := FALSE; END_IF;
END_REGION
END_FUNCTION_BLOCK

FUNCTION_BLOCK "ALARMS_SCL"   // FB13, SCL
{ S7_Optimized_Access := 'TRUE' }
VERSION : 0.1
   VAR_TEMP
      t1 : Time;
      tm1 : Time;
      OFLAT : Bool;
      tm2 : Time;
      OCAT : Bool;
      t2 : Time;
      tm3 : Time;
      tm4 : Time;
      tm5 : Time;
      tm6 : Time;
      tm7 : Time;
      t3 : Time;
      t4 : Time;
      t5 : Time;
      t6 : Time;
      t7 : Time;
      HOTAT : Bool;
      ROAT : Bool;
      OHFAT : Bool;
      BFAT : Bool;
      ESAT : Int;
   END_VAR
BEGIN
   // Oil Low Flow Alarm
   IF "OilPumpVFDen_Out" AND "OilFlow" < "OilLLFlow_Sp"  AND NOT "Brake_Out" AND NOT "OilLowFlowAlarm" AND NOT "AlarmReset" THEN
   "CONVERTTIME"(Int1:="OilLowFlowDelay_Sp",
                 tem1=>#tm1);

       "IEC_Timer_0_DB_12".TON(IN := TRUE,
                               PT := #tm1,
                               Q => #OFLAT,
                               ET => #t1);

   END_IF;

   IF #OFLAT THEN
       "OilLowFlowAlarm" := 1;
       "OilLowFlowNotify" := 1;
   END_IF;

   IF "OilLowFlowAlarm" AND "AlarmReset" THEN
       "OilLowFlowAlarm" := 0;
       "OilLowFlowNotify" := 0;
   END_IF;

   IF "OilLowFlowNotify" AND "AlarmSilence" THEN
       "OilLowFlowNotify" := 0;
   END_IF;

   // Over Current Alarm
   IF "Current" < "OverCurrent_Sp" AND NOT "AlarmReset" AND NOT "OverCurrentAlarm" THEN
       "CONVERTTIME"(Int1 := "OverCurrentDelay_Sp",
                     tem1 => #tm2);
       "IEC_Timer_0_DB_13".TON(IN := TRUE,
                               PT := #tm2,
                               Q => #OCAT,
                               ET => #t2);

   END_IF;

   IF #OCAT THEN
       "OverCurrentAlarm" := 1;
       "OverCurrentNotify" := 1;
   END_IF;

   IF #OCAT AND "AlarmReset" THEN
       "OverCurrentAlarm" := 0;
       "OverCurrentNotify" := 0;
   END_IF;

   IF "OverCurrentNotify" AND "AlarmSilence" THEN
       "OverCurrentNotify" := 0;
   END_IF;

   // High Oil Temp Alarm

   IF "OilTemp" > "HighOilTemp _Sp" AND NOT "OilTempAlarm" AND NOT "OilTempAlarmNotify" THEN
       "CONVERTTIME"(Int1 := "OilHighFlowDelay_Sp",
                     tem1 => #tm3);
       "IEC_Timer_0_DB_14".TON(IN := TRUE,
                               PT := #tm3,
                               Q => #HOTAT,
                               ET => #t3);
   END_IF;

   IF #HOTAT AND "AlarmReset" THEN
       "OilTempAlarm" := 0;
       "OilTempAlarmNotify" := 0;
   END_IF;

   IF #HOTAT THEN
       "OilTempAlarm" := 1;
       "OilTempAlarmNotify" := 1;
   END_IF;

   IF "OilTempAlarmNotify" AND "AlarmSilence" THEN
       "OilTempAlarmNotify" := 0;
   END_IF;

   // RottorOverspeed 

   IF "RPM" > "RottorOverspeed_Sp" AND NOT "AlarmReset" AND NOT "RottorOverspeedAlarm" THEN
       "CONVERTTIME"(Int1 := "RottorOverspeedDelay_Sp",
                     tem1 => #tm4);
       "IEC_Timer_0_DB_13".TON(IN := TRUE,
                               PT := #tm4,
                               Q => #ROAT,
                               ET => #t4);

   END_IF;


       IF #OCAT THEN
           "RottorOverspeedAlarm" := 1;
           "RottorOverspeedNotify" := 1;
       END_IF;

       IF #OCAT AND "AlarmReset" THEN
           "RottorOverspeedAlarm" := 0;
           "RottorOverspeedNotify" := 0;
       END_IF;

       IF "RottorOverspeedNotify" AND "AlarmSilence" THEN
           "RottorOverspeedNotify" := 0;
       END_IF;

   // OIL High Flow Alarm


       IF "OilFlow" > "OilHHFlow_Sp" AND NOT "AlarmReset" AND NOT "OilHighFlowAlarm" THEN
           "CONVERTTIME"(Int1 := "OilHighFlowDelay_Sp",
                     tem1 => #tm5);
       "IEC_Timer_0_DB_13".TON(IN := TRUE,
                               PT := #tm5,
                               Q => #OHFAT,
                               ET => #t5);

   END_IF;


   IF #OHFAT THEN
       "OilHighFlowAlarm" := 1;
       "OilHighFlowNotify" := 1;
   END_IF;

   IF #OHFAT AND "AlarmReset" THEN
       "OilHighFlowAlarm" := 0;
       "OilHighFlowNotify" := 0;
   END_IF;

   IF "OilHighFlowNotify" AND "AlarmSilence" THEN
       "OilHighFlowNotify" := 0;
   END_IF;

   // Brake Failuer Alarm



   IF "RPM" > 0 AND "Brake_Out" AND NOT "AlarmReset" AND NOT "BrakeFalierAlarm" THEN
       "CONVERTTIME"(Int1 := "BraheFailuerDelay_Sp",
                     tem1 => #tm6);
       "IEC_Timer_0_DB_13".TON(IN := TRUE,
                               PT := #tm6,
                               Q => #BFAT,
                               ET => #t6);

   END_IF;


   IF #BFAT THEN
       "BrakeFalierAlarm" := 1;
       "BrakeFalierAlarmNotify" := 1;
   END_IF;

   IF #BFAT AND "AlarmReset" THEN
       "BrakeFalierAlarm" := 0;
       "BrakeFalierAlarmNotify" := 0;
   END_IF;

   IF "BrakeFalierAlarmNotify" AND "AlarmSilence" THEN
       "BrakeFalierAlarmNotify" := 0;
   END_IF;

   // EStop

   IF "EStop" AND NOT "AlarmReset" THEN
       "EStaoAlarm" := 1;
       "EStapAlarmNotify" := 1;
   END_IF;

   IF "EStaoAlarm" AND "AlarmReset" THEN
       "EStaoAlarm" := 0;
       "EStapAlarmNotify" := 0;
   END_IF;

   IF "EStapAlarmNotify" AND "AlarmSilence" THEN
       "EStapAlarmNotify" := 0;
   END_IF;
END_FUNCTION_BLOCK

FUNCTION_BLOCK "ALARMS_STL"   // FB14, STL
{ S7_Optimized_Access := 'TRUE' }
VERSION : 0.1
   VAR
      OS1 : Bool;
      OS2 : Bool;
   END_VAR
   VAR_TEMP
      ti1 : Time;
      t1 : Time;
      OLFAT : Bool;
   END_VAR
BEGIN

REGION Network 1
   // Oil Low Flow Alarm
         L     "OilFlow";
         L     "OilHHFlow_Sp";
         <I;
         A     "OilPumpVFDen_Out";
         AN    "Brake_Out";
         JC    OLFtimer;
         CLR;
         A     "AlarmReset";
         FP    #OS1;
         A     "AlarmSilence";
         FP    #OS2;
         JC    ResetOLFnotify;


   OLFtimer:CALL  "CONVERTTIME"
         ( Int1 := "OilLowFlowDelay_Sp",
           tem1 := #ti1
         );
         CALL  TON, "IEC_Timer_0_DB_15"
         ( IN := TRUE,
           PT := #ti1,
           Q  := #OLFAT,
           ET := #t1
         );
         A     #OLFAT;
         JC    SetOLFalarm;
         JU    Endofline;

   SetOLFalarm:SET;
         S     "OilLowFlowAlarm";
         S     "OilLowFlowNotify";
         JU    Endofline;
   ResetOLFalarm:R     "OilLowFlowAlarm";
         R     "OilLowFlowNotify";
   ResetOLFnotify:R     "OilLowFlowNotify";
         JU    Endofline;

   Endofline:BE;

   //
END_REGION
END_FUNCTION_BLOCK

FUNCTION_BLOCK "MODES_LAD"   // FB15, LAD
{ S7_Optimized_Access := 'TRUE' }
VERSION : 0.1
// Modes:
// Warmup
//  – When Start pushbutton is pressed, the sequence begins with this step. Allow the rotor to 
// turn at a speed somethere between 20 and 50 RPMs and run the oil pump at some low output level (2-
// 10 GPM maybe?) until the oil temp reaches 150 degrees. Once we’ve maintained at least 150 degrees 
// for 10 seconds, we want to transition into the next mode.
// (continued)
// Stabiliz
// e – Generator should speed up until desired kW output is attained. Once we’re stable within 
// 5kW (+/-) of the setpoint for at least 10 seconds, we should transition into the next mode. 
// Generation
//  – Keep everything running and close the interlock.
// Cooldown
//  – Once the Stop button has been pushed, open the interlock, slow the rotor to between 20 
// and 50 RPMs and maintain a high oil flow until the oil temp is below 150 degrees. Once we’re below 
// for ten seconds, we transition into Idle mode.
// Idle – Interlock and baffle are deenergized and brake is engaged.
// Fault
//  – When we hit an alarm, the sequence should be aborted according to the alarm details (above in 
// the Alarms section), and we should go into Fault mode (which is not part of our sequence)
   VAR
      os1 : Bool;
      os2 : Bool;
      os3 : Bool;
      os4 : Bool;
      os5 : Bool;
   END_VAR
   VAR_TEMP
      tv1 : Int;
      ti1 : Time;
      tv2 : Int;
      tv3 : Int;
      tv4 : Int;
      ti2 : Time;
      tv5 : Int;
      ti3 : Time;
   END_VAR
   VAR_TEMP   // added for the SCL form of the ladder/FBD networks
      _w1 : Bool;
      _w2 : Bool;
      _w3 : Bool;
   END_VAR
BEGIN

REGION Network 1
   // Wormup Mode
   // Warmup
   //  – When Start pushbutton is pressed, the sequence begins with this step. Allow the rotor to 
   // turn at a speed somethere between 20 and 50 RPMs and run the oil pump at some low output level (2-
   // 10 GPM maybe?) until the oil temp reaches 150 degrees. Once we’ve maintained at least 150 degrees 
   // for 10 seconds, we want to transition into the next mode.
   // (continued)
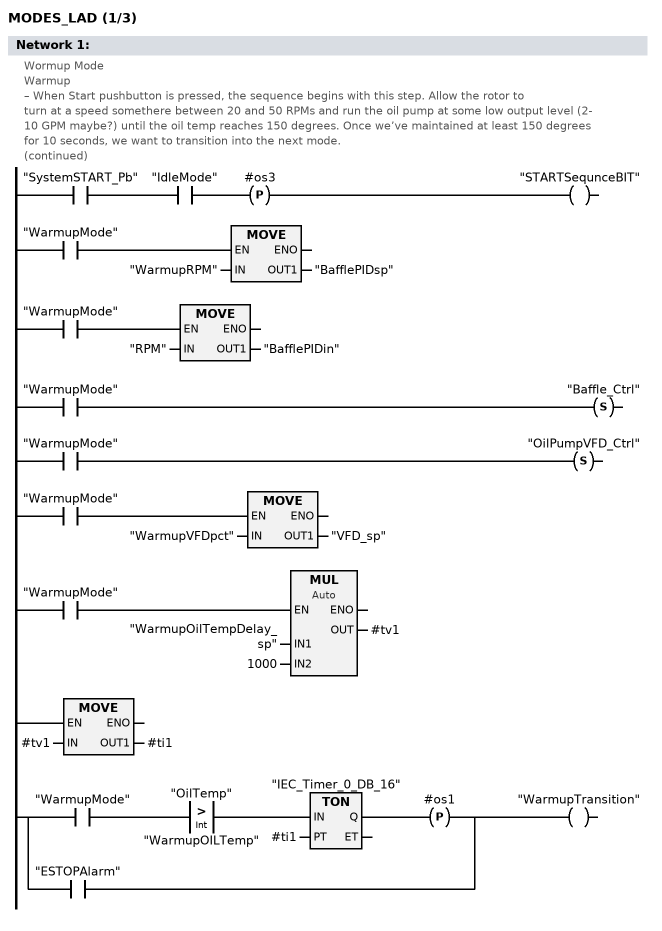
   #_w1 := "SystemSTART_Pb" AND "IdleMode";
   #_w2 := #_w1 AND NOT #os3;   // rising edge
   #os3 := #_w1;
   "STARTSequnceBIT" := #_w2;
   IF "WarmupMode" THEN
       "BafflePIDsp" := "WarmupRPM";
       "BafflePIDin" := "RPM";
       "Baffle_Ctrl" := TRUE;
       "OilPumpVFD_Ctrl" := TRUE;
       "VFD_sp" := "WarmupVFDpct";
       #tv1 := "WarmupOilTempDelay_sp" * 1000;
   END_IF;
   #ti1 := #tv1;
   "IEC_Timer_0_DB_16".TON(IN := "WarmupMode" AND ("OilTemp" > "WarmupOILTemp"), PT := #ti1);
   #_w3 := "IEC_Timer_0_DB_16".Q AND NOT #os1;   // rising edge
   #os1 := "IEC_Timer_0_DB_16".Q;
   "WarmupTransition" := #_w3 OR "ESTOPAlarm";
END_REGION

REGION Network 2
   // Stabilize Mode
   // Stabiliz
   // e – Generator should speed up until desired kW output is attained. Once we’re stable within 
   // 5kW (+/-) of the setpoint for at least 10 seconds, we should transition into the next mode.
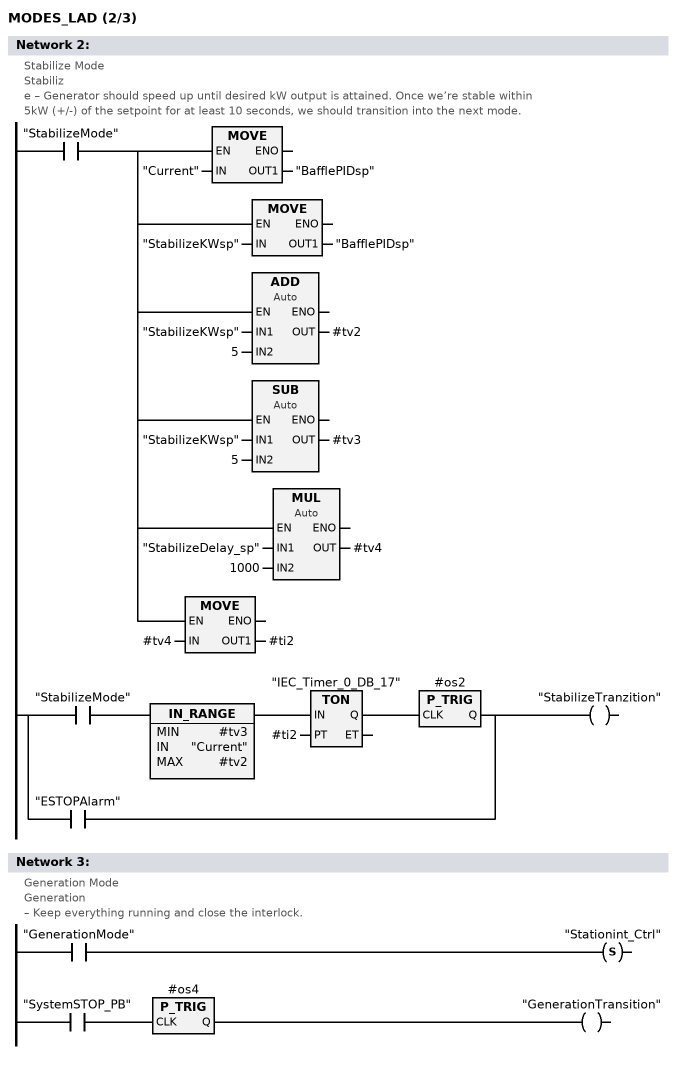
   IF "StabilizeMode" THEN
       "BafflePIDsp" := "Current";
       "BafflePIDsp" := "StabilizeKWsp";
       #tv2 := "StabilizeKWsp" + 5;
       #tv3 := "StabilizeKWsp" - 5;
       #tv4 := "StabilizeDelay_sp" * 1000;
       #ti2 := #tv4;
   END_IF;
   "IEC_Timer_0_DB_17".TON(IN := "StabilizeMode" AND (#tv3 <= "Current") AND ("Current" <= #tv2), PT := #ti2);
   #_w1 := "IEC_Timer_0_DB_17".Q AND NOT #os2;   // rising edge
   #os2 := "IEC_Timer_0_DB_17".Q;
   "StabilizeTranzition" := #_w1 OR "ESTOPAlarm";
END_REGION

REGION Network 3
   // Generation Mode
   // Generation
   //  – Keep everything running and close the interlock.
   RUNG wire#powerrail
      Contact( "GenerationMode" )
      S_Coil( "Stationint_Ctrl" )
   END_RUNG
   RUNG wire#powerrail
      Contact( "SystemSTOP_PB" )
      P_Trig( #os4 )
      Coil( "GenerationTransition" )
   END_RUNG
   // the same network as SCL:
   IF "GenerationMode" THEN "Stationint_Ctrl" := TRUE; END_IF;
   #_w1 := "SystemSTOP_PB" AND NOT #os4;   // rising edge
   #os4 := "SystemSTOP_PB";
   "GenerationTransition" := #_w1;
END_REGION

REGION Network 4
   // Cooldown Mode
   // Cooldown
   //  – Once the Stop button has been pushed, open the interlock, slow the rotor to between 20 
   // and 50 RPMs and maintain a high oil flow until the oil temp is below 150 degrees. Once we’re below 
   // for ten seconds, we transition into Idle mode.
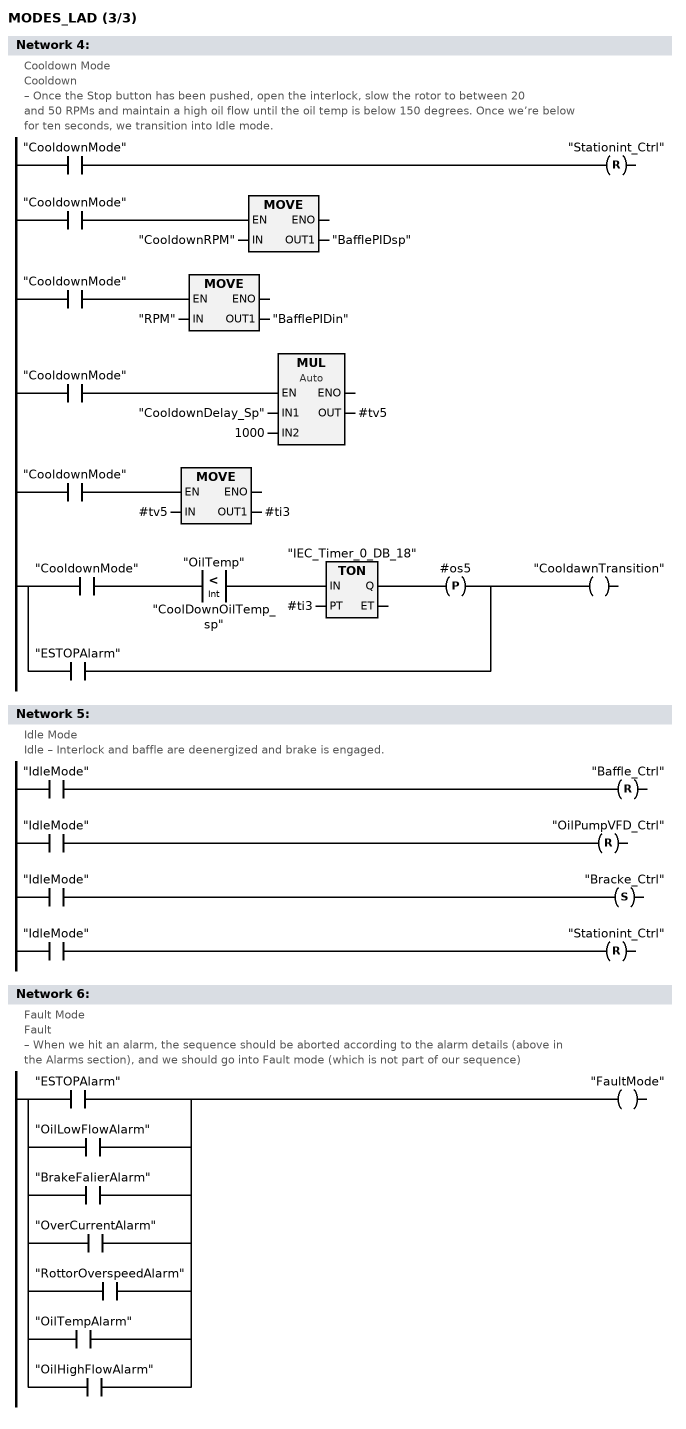
   IF "CooldownMode" THEN
       "Stationint_Ctrl" := FALSE;
       "BafflePIDsp" := "CooldownRPM";
       "BafflePIDin" := "RPM";
       #tv5 := "CooldownDelay_Sp" * 1000;
       #ti3 := #tv5;
   END_IF;
   "IEC_Timer_0_DB_18".TON(IN := "CooldownMode" AND ("OilTemp" < "CoolDownOilTemp_sp"), PT := #ti3);
   #_w1 := "IEC_Timer_0_DB_18".Q AND NOT #os5;   // rising edge
   #os5 := "IEC_Timer_0_DB_18".Q;
   "CooldawnTransition" := #_w1 OR "ESTOPAlarm";
END_REGION

REGION Network 5
   // Idle Mode 
   // Idle – Interlock and baffle are deenergized and brake is engaged.
   RUNG wire#powerrail
      Contact( "IdleMode" )
      R_Coil( "Baffle_Ctrl" )
   END_RUNG
   RUNG wire#powerrail
      Contact( "IdleMode" )
      R_Coil( "OilPumpVFD_Ctrl" )
   END_RUNG
   RUNG wire#powerrail
      Contact( "IdleMode" )
      S_Coil( "Bracke_Ctrl" )
   END_RUNG
   RUNG wire#powerrail
      Contact( "IdleMode" )
      R_Coil( "Stationint_Ctrl" )
   END_RUNG
   // the same network as SCL:
   IF "IdleMode" THEN
       "Baffle_Ctrl" := FALSE;
       "OilPumpVFD_Ctrl" := FALSE;
       "Bracke_Ctrl" := TRUE;
       "Stationint_Ctrl" := FALSE;
   END_IF;
END_REGION

REGION Network 6
   // Fault Mode 
   // Fault
   //  – When we hit an alarm, the sequence should be aborted according to the alarm details (above in 
   // the Alarms section), and we should go into Fault mode (which is not part of our sequence)
   RUNG wire#powerrail
      Contact( "ESTOPAlarm" )
      wire#w1
      Coil( "FaultMode" )
   END_RUNG
   RUNG wire#powerrail
      Contact( "OilLowFlowAlarm" )
   END_RUNG wire#w1
   RUNG wire#powerrail
      Contact( "BrakeFalierAlarm" )
   END_RUNG wire#w1
   RUNG wire#powerrail
      Contact( "OverCurrentAlarm" )
   END_RUNG wire#w1
   RUNG wire#powerrail
      Contact( "RottorOverspeedAlarm" )
   END_RUNG wire#w1
   RUNG wire#powerrail
      Contact( "OilTempAlarm" )
   END_RUNG wire#w1
   RUNG wire#powerrail
      Contact( "OilHighFlowAlarm" )
   END_RUNG wire#w1
   // the same network as SCL:
   "FaultMode" := "ESTOPAlarm" OR "OilLowFlowAlarm" OR "BrakeFalierAlarm" OR "OverCurrentAlarm" OR "RottorOverspeedAlarm" OR "OilTempAlarm" OR "OilHighFlowAlarm";
END_REGION
END_FUNCTION_BLOCK

FUNCTION_BLOCK "MODES_FBD"   // FB16, FBD
{ S7_Optimized_Access := 'TRUE' }
VERSION : 0.1
   VAR
      OS1 : Bool;
      OS2 : Bool;
      OS3 : Bool;
      OS4 : Bool;
      OS5 : Bool;
   END_VAR
   VAR_TEMP
      ti1 : Time;
      tv1 : Int;
      tv2 : Int;
      ti3 : Time;
      ti4 : Time;
   END_VAR
   VAR_TEMP   // added for the SCL form of the ladder/FBD networks
      _w1 : Bool;
      _w2 : Bool;
      _w3 : Bool;
   END_VAR
BEGIN

REGION Network 1
   // Warmup
   //  – When Start pushbutton is pressed, the sequence begins with this step. Allow the rotor to 
   // turn at a speed somethere between 20 and 50 RPMs and run the oil pump at some low output level (2-
   // 10 GPM maybe?) until the oil temp reaches 150 degrees. Once we’ve maintained at least 150 degrees 
   // for 10 seconds, we want to transition into the next mode.
   // (continued)
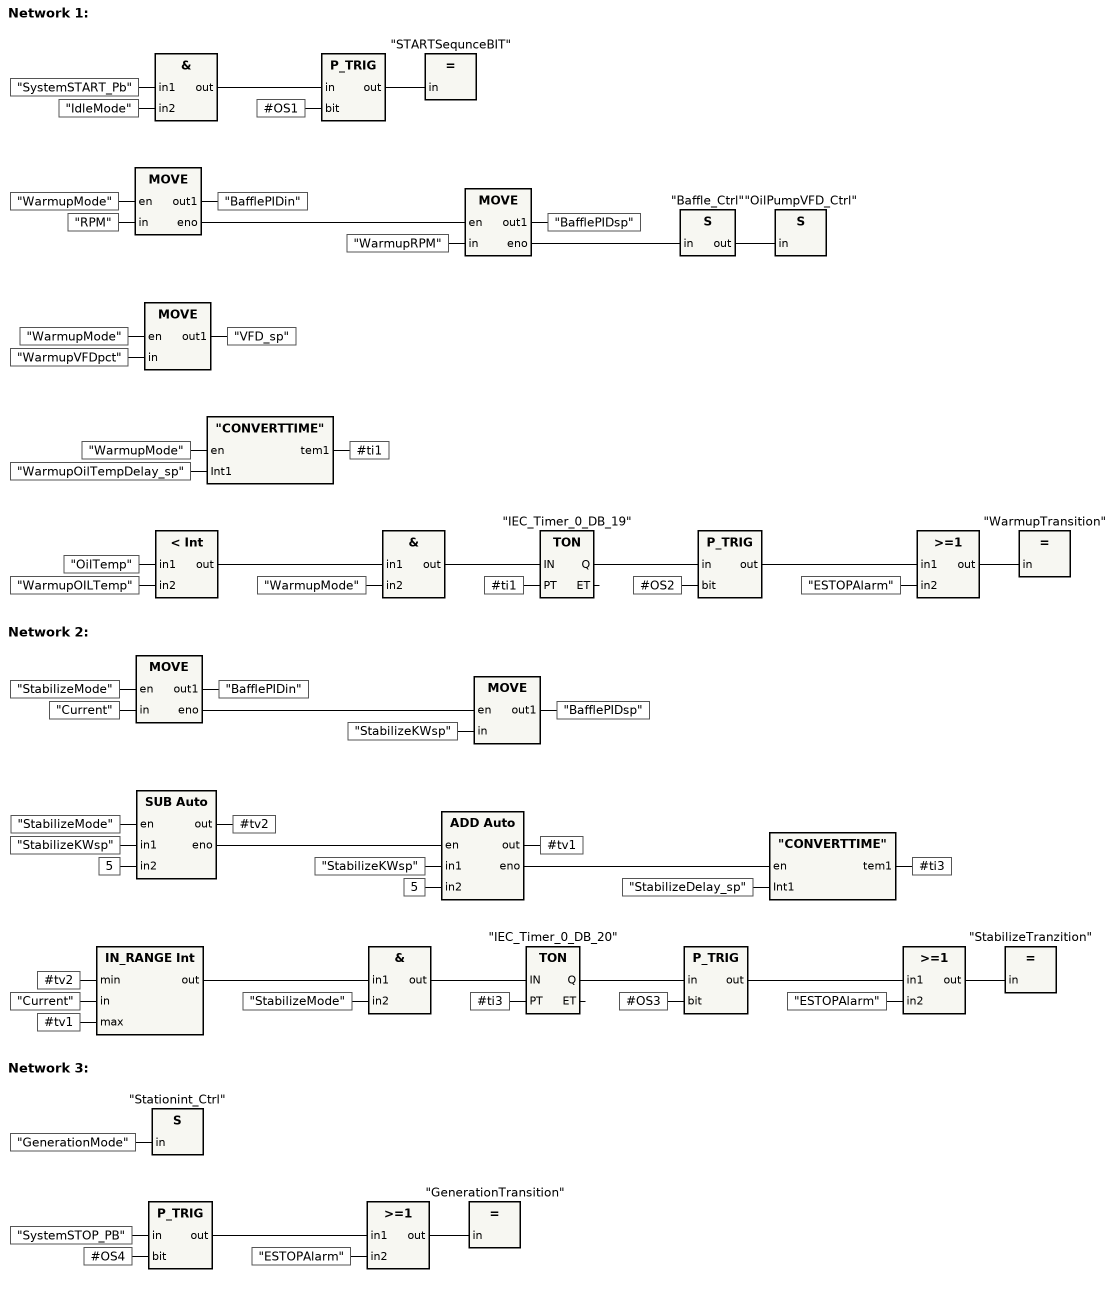
   #_w1 := "SystemSTART_Pb" AND "IdleMode";
   #_w2 := #_w1 AND NOT #OS1;   // rising edge
   #OS1 := #_w1;
   "STARTSequnceBIT" := #_w2;
   IF "WarmupMode" THEN
       "BafflePIDin" := "RPM";
       "BafflePIDsp" := "WarmupRPM";
       "Baffle_Ctrl" := TRUE;
       "OilPumpVFD_Ctrl" := TRUE;
       "VFD_sp" := "WarmupVFDpct";
       "CONVERTTIME"(Int1 := "WarmupOilTempDelay_sp", tem1 => #ti1);
   END_IF;
   "IEC_Timer_0_DB_19".TON(IN := ("OilTemp" < "WarmupOILTemp") AND "WarmupMode", PT := #ti1);
   #_w3 := "IEC_Timer_0_DB_19".Q AND NOT #OS2;   // rising edge
   #OS2 := "IEC_Timer_0_DB_19".Q;
   "WarmupTransition" := #_w3 OR "ESTOPAlarm";
END_REGION

REGION Network 2
   // STabilize Mode
   // Stabiliz
   // e – Generator should speed up until desired kW output is attained. Once we’re stable within 
   // 5kW (+/-) of the setpoint for at least 10 seconds, we should transition into the next mode.
   IF "StabilizeMode" THEN
       "BafflePIDin" := "Current";
       "BafflePIDsp" := "StabilizeKWsp";
       #tv2 := "StabilizeKWsp" - 5;
       #tv1 := "StabilizeKWsp" + 5;
       "CONVERTTIME"(Int1 := "StabilizeDelay_sp", tem1 => #ti3);
   END_IF;
   "IEC_Timer_0_DB_20".TON(IN := (#tv2 <= "Current") AND ("Current" <= #tv1) AND "StabilizeMode", PT := #ti3);
   #_w1 := "IEC_Timer_0_DB_20".Q AND NOT #OS3;   // rising edge
   #OS3 := "IEC_Timer_0_DB_20".Q;
   "StabilizeTranzition" := #_w1 OR "ESTOPAlarm";
END_REGION

REGION Network 3
   // Generation Mode
   // Generation
   //  – Keep everything running and close the interlock.
   IF "GenerationMode" THEN "Stationint_Ctrl" := TRUE; END_IF;
   #_w1 := "SystemSTOP_PB" AND NOT #OS4;   // rising edge
   #OS4 := "SystemSTOP_PB";
   "GenerationTransition" := #_w1 OR "ESTOPAlarm";
END_REGION

REGION Network 4
   // Cooldown Mode
   // Cooldown
   //  – Once the Stop button has been pushed, open the interlock, slow the rotor to between 20 
   // and 50 RPMs and maintain a high oil flow until the oil temp is below 150 degrees. Once we’re below 
   // for ten seconds, we transition into Idle mode.
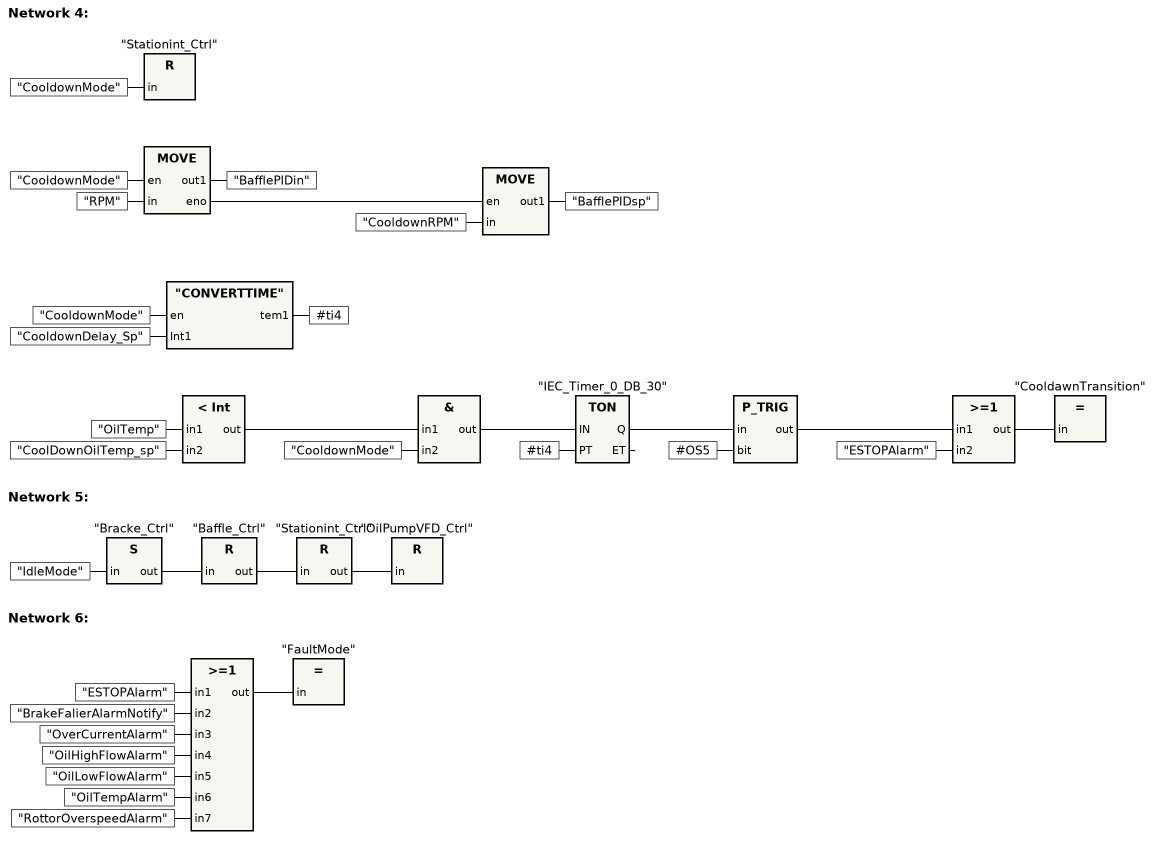
   IF "CooldownMode" THEN
       "Stationint_Ctrl" := FALSE;
       "BafflePIDin" := "RPM";
       "BafflePIDsp" := "CooldownRPM";
       "CONVERTTIME"(Int1 := "CooldownDelay_Sp", tem1 => #ti4);
   END_IF;
   "IEC_Timer_0_DB_30".TON(IN := ("OilTemp" < "CoolDownOilTemp_sp") AND "CooldownMode", PT := #ti4);
   #_w1 := "IEC_Timer_0_DB_30".Q AND NOT #OS5;   // rising edge
   #OS5 := "IEC_Timer_0_DB_30".Q;
   "CooldawnTransition" := #_w1 OR "ESTOPAlarm";
END_REGION

REGION Network 5
   // dle Mode 
   // Idle – Interlock and baffle are deenergized and brake is engaged.
   IF "IdleMode" THEN
       "Bracke_Ctrl" := TRUE;
       "Baffle_Ctrl" := FALSE;
       "Stationint_Ctrl" := FALSE;
       "OilPumpVFD_Ctrl" := FALSE;
   END_IF;
END_REGION

REGION Network 6
   // Fault Mode 
   // Fault
   //  – When we hit an alarm, the sequence should be aborted according to the alarm details (above in 
   // the Alarms section), and we should go into Fault mode (which is not part of our sequence)
   "FaultMode" := "ESTOPAlarm" OR "BrakeFalierAlarmNotify" OR "OverCurrentAlarm" OR "OilHighFlowAlarm" OR "OilLowFlowAlarm" OR "OilTempAlarm" OR "RottorOverspeedAlarm";
END_REGION
END_FUNCTION_BLOCK

FUNCTION_BLOCK "SEQUENCE"   // FB17, GRAPH_PLUS
{ S7_Optimized_Access := 'TRUE' }
VERSION : 0.1
   VAR_INPUT
      OFF_SQ : Bool := false;   // Turn sequence off
      INIT_SQ : Bool := false;   // Set sequence to initial state
      ACK_EF : Bool := false;   // Acknowledge all errors and faults
      S_PREV : Bool := false;   // Output previous step in parameter S_NO
      S_NEXT : Bool := false;   // Indicate next step in parameter S_NO
      SW_AUTO : Bool := false;   // Automatic mode
      SW_TAP : Bool := false;   // Semiautomatic/switch with transition
      SW_TOP : Bool := false;   // Semiautomatic/ignore transition
      SW_MAN : Bool := false;   // Manual mode
      S_SEL : Int := 0;   // Select step to be output to S_NO
      S_ON : Bool := false;   // Activate step indicated in S_NO
      S_OFF : Bool := false;   // Deactivate step indicated S_NO
      T_PUSH : Bool := false;   // Enable transition to switch in semi automatic mode
   END_VAR
   VAR_OUTPUT
      S_NO : Int := 0;   // Step number
      S_MORE : Bool := false;   // More steps are available and can be shown in S_NO
      S_ACTIVE : Bool := false;   // Step indicated in S_NO is active
      ERR_FLT : Bool := false;   // Interlock or supervision group error
      AUTO_ON : Bool := false;   // Automatic mode is active
      TAP_ON : Bool := false;   // Semiautomatic mode/step with transition enabled
      TOP_ON : Bool := false;   // Semiautomatic mode/ignore transition enabled
      MAN_ON : Bool := false;   // Manual mode is active
   END_VAR
   VAR
      HMI_INFO : Array[0..8] of UInt;
      IF_PAR : G7_IfParPlus_V2;
      RT_DATA : G7_RTDataPlus_V2;   // Internal data area
      Trans1 : G7_TransitionPlus_V2;   // Transition structure
      Trans2 : G7_TransitionPlus_V2;   // Transition structure
      Trans3 : G7_TransitionPlus_V2;   // Transition structure
      Trans4 : G7_TransitionPlus_V2;   // Transition structure
      Trans5 : G7_TransitionPlus_V2;   // Transition structure
      Idle : G7_StepPlus_V2;   // Step structure
      Warmup : G7_StepPlus_V2;   // Step structure
      Stabilize : G7_StepPlus_V2;   // Step structure
      Generation : G7_StepPlus_V2;   // Step structure
      Cooldown : G7_StepPlus_V2;   // Step structure
      SINI : Array[0..1] of USInt;
      LSTT : Array[0..4] of USInt;
      ATAJ : Array[0..4] of USInt;
      ATAB : Array[0..4] of USInt;
      PSTT : Array[0..4] of USInt;
      NSTT : Array[0..4] of USInt;
      ASSJ : Array[0..4] of USInt;
      ASSB : Array[0..4] of USInt;
      PTTS : Array[0..4] of USInt;
      NTTS : Array[0..4] of USInt;
      SW_SQTS : Array[0..4] of USInt;
      SWITCH : Array[0..0] of USInt;
      TVX : Array[0..1] of USInt;
      TTX : Array[0..1] of USInt;
      TSX : Array[0..1] of USInt;
      S00X : Array[0..1] of USInt;
      SOFFX : Array[0..1] of USInt;
      SONX : Array[0..1] of USInt;
      SAX : Array[0..1] of USInt;
      SERRX : Array[0..5] of USInt;
      SMX : Array[0..5] of USInt;
      S0X : Array[0..5] of USInt;
      S1X : Array[0..5] of USInt;
      IL_ALARM_INST : Program_Alarm;
      SUP_ALARM_INST : Program_Alarm;
      STEP_TIME_ALARM_INST : Program_Alarm;
      IEC_TIMER_INST : IEC_TIMER;
      TRANSACTION_FLAG : Bool := false;
   END_VAR
   // SINI[0] := 2;
   // SINI[1] := 1;
   // LSTT[0] := 255;
   // LSTT[1] := 255;
   // LSTT[2] := 255;
   // LSTT[3] := 255;
   // ATAJ[1] := 1;
   // ATAJ[2] := 2;
   // ATAJ[3] := 3;
   // ATAJ[4] := 4;
   // ATAB[1] := 1;
   // ATAB[2] := 2;
   // ATAB[3] := 3;
   // ATAB[4] := 4;
   // PSTT[1] := 1;
   // PSTT[2] := 2;
   // PSTT[3] := 3;
   // PSTT[4] := 4;
   // NSTT[0] := 1;
   // NSTT[1] := 2;
   // NSTT[2] := 3;
   // NSTT[3] := 4;
   // ASSJ[1] := 1;
   // ASSJ[2] := 2;
   // ASSJ[3] := 3;
   // ASSJ[4] := 4;
   // ASSB[1] := 1;
   // ASSB[2] := 2;
   // ASSB[3] := 3;
   // ASSB[4] := 4;
   // PTTS[0] := 255;
   // PTTS[2] := 1;
   // PTTS[3] := 2;
   // PTTS[4] := 3;
   // NTTS[1] := 1;
   // NTTS[2] := 2;
   // NTTS[3] := 3;
   // NTTS[4] := 4;
   // TVX[0] := 16#1;
   // TTX[0] := 16#1;
   // TSX[0] := 16#1;
   // S00X[0] := 16#1;
   // SOFFX[0] := 16#1;
   // SONX[0] := 16#1;
   // SAX[0] := 16#1;
   // SERRX[0] := 16#1;
   // SMX[0] := 16#1;
   // S0X[0] := 16#1;
   // S1X[0] := 16#1;
BEGIN
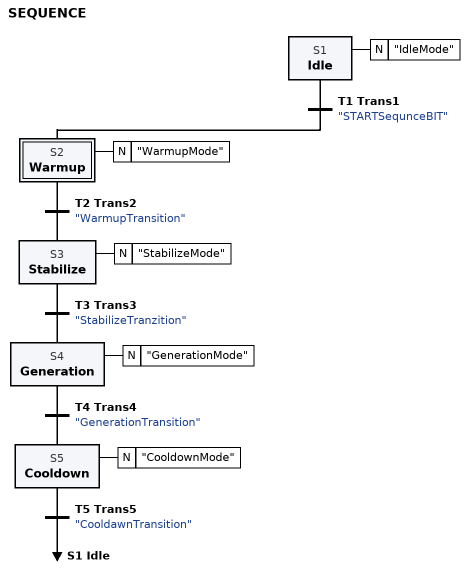
   // sequencer 1
   STEP Idle:   // S1, max time T#10S, warning time T#7S
              N    "IdleMode"
   END_STEP
   TRANSITION Trans1 FROM Idle TO Warmup   // T1
      := "STARTSequnceBIT";
   END_TRANSITION
   INITIAL_STEP Warmup:   // S2, max time T#10S, warning time T#7S
              N    "WarmupMode"
   END_STEP
   TRANSITION Trans2 FROM Warmup TO Stabilize   // T2
      := "WarmupTransition";
   END_TRANSITION
   STEP Stabilize:   // S3, max time T#10S, warning time T#7S
              N    "StabilizeMode"
   END_STEP
   TRANSITION Trans3 FROM Stabilize TO Generation   // T3
      := "StabilizeTranzition";
   END_TRANSITION
   STEP Generation:   // S4, max time T#10S, warning time T#7S
              N    "GenerationMode"
   END_STEP
   TRANSITION Trans4 FROM Generation TO Cooldown   // T4
      := "GenerationTransition";
   END_TRANSITION
   STEP Cooldown:   // S5, max time T#10S, warning time T#7S
              N    "CooldownMode"
   END_STEP
   TRANSITION Trans5 FROM Cooldown TO Idle   // T5, jump
      := "CooldawnTransition";
   END_TRANSITION
END_FUNCTION_BLOCK

FUNCTION_BLOCK "MODES_SCL"   // FB18, SCL
{ S7_Optimized_Access := 'TRUE' }
VERSION : 0.1
   VAR_TEMP
      warmupdelaytrigger_1 : Bool;
      ti1 : Time;
      ti2 : Time;
      tv1 : Int;
      tv2 : Int;
      ti3 : Time;
      stabilizedelaytreagger : Bool;
      ti4 : Time;
      warmupdelaytrigger : Bool;
      ti5 : Time;
      cooldowdelaytreggar : Bool;
      ti6 : Time;
   END_VAR
BEGIN
   // Wormup Mode
   //Warmup
   //– When Start pushbutton is pressed, the sequence begins with this step. Allow the rotor TO
   //turn at a speed somethere between 20 AND 50 RPMs AND run the oil pump at some low output level (2-
   //10 GPM maybe?) UNTIL the oil temp reaches 150 degrees. Once we’ve maintained at least 150 degrees
   //FOR 10 seconds, we want TO transition into the next mode.
   //
   IF "SystemSTART_Pb" AND "IdleMode" THEN
       "STARTSequnceBIT" := 1;
   ELSE
       "STARTSequnceBIT" := 0;
   END_IF;

   IF "WarmupMode" THEN
       "BafflePIDin" := "RPM";
       "BafflePIDsp" := "WarmupRPM";
       "VFD_sp" := "WarmupVFDpct";
       IF "OilTemp" > "WarmupOILTemp" THEN
           "CONVERTTIME"(Int1 := "WarmupOilTempDelay_sp",
                         tem1 => #ti1);

           "IEC_Timer_0_DB_22".TON(IN := TRUE,
                                   PT := #ti1,
                                   Q => #warmupdelaytrigger,
                                   ET => #ti2);
       ELSE
           RESET_TIMER("IEC_Timer_0_DB_22");

       END_IF;

       IF #warmupdelaytrigger THEN
           RESET_TIMER("IEC_Timer_0_DB_22");
           "WarmupTransition" := 1;
       END_IF;
   ELSE
       "WarmupTransition" := 0;
   END_IF;


   // Stabilaze Mode 
   // 

   IF "StabilizeMode" THEN
       "BafflePIDin" := "Current";
       "BafflePIDsp" := "StabilizeKWsp";
       #tv1 := "StabilizeKWsp" - 5;
       #tv2 := "StabilizeKWsp" + 5;
       IF "Current" < #tv2 AND "Current" > #tv1 THEN
           "CONVERTTIME"(Int1 := "StabilizeDelay_sp",
                         tem1 => #ti3);
           "IEC_Timer_0_DB_23".TON(IN := TRUE,
                                   PT := #ti3,
                                   Q => #stabilizedelaytreagger,
                                   ET => #ti4);
       ELSE
           RESET_TIMER("IEC_Timer_0_DB_23");
       END_IF;
       IF #stabilizedelaytreagger THEN
           "StabilizeTranzition" := 1;
       END_IF;
   ELSE
       "StabilizeTranzition" := 0;
   END_IF;

   // generation Mode
   // 
   IF "GenerationMode" THEN
       "Stationint_Ctrl" := 1;
       IF "SystemSTOP_PB" THEN
           "GenerationTransition" := 1;
       END_IF;
   ELSE
       "GenerationTransition" := 0;
   END_IF;

   // Cooldown Mode 
   // 
   IF "CooldownMode" THEN
       "Stationint_Ctrl" := 0;
       "BafflePIDin" := "RPM";
       "BafflePIDsp" := "CoolDownRPM_sp";
       IF "OilTemp" < "CoolDownOilTemp_sp" THEN
           "CONVERTTIME"(Int1 := "CooldownDelay_Sp",
                         tem1 => #ti5);
           "IEC_Timer_0_DB_24".TON(IN := TRUE,
                                   PT := #ti5,
                                   Q => #cooldowdelaytreggar,
                                   ET => #ti6);
       ELSE
           RESET_TIMER("IEC_Timer_0_DB_24");
       END_IF;
       IF #cooldowdelaytreggar THEN
           RESET_TIMER("IEC_Timer_0_DB_24");
           "CooldawnTransition" := 1;
       END_IF;
   ELSE
       "CooldawnTransition" := 0;
   END_IF;

   // Idel Mode 
   // 
   IF "IdleMode" THEN
       "Bracke_Ctrl" := 1;
       "OilPumpVFD_Ctrl" := 0;
       "Baffle_Ctrl" := 0;
       "Stationint_Ctrl" := 0;
   END_IF;

   // Fault Mode
   // 
   IF "ESTOPAlarm" OR "BrakeFalierAlarm" OR "OverCurrentAlarm" OR "RottorOverspeedAlarm" OR "OilLowFlowAlarm" OR "OilHighFlowAlarm" OR "OilTempAlarm" THEN
       "FaultMode" := 1;
   ELSE
       "FaultMode" := 0;
   END_IF;
END_FUNCTION_BLOCK

FUNCTION_BLOCK "MODE_STL"   // FB19, STL
{ S7_Optimized_Access := 'TRUE' }
VERSION : 0.1
   VAR
      OS1 : Bool;
   END_VAR
   VAR_TEMP
      ti1 : Time;
      warmupdelaytrigger : Bool;
      ti2 : Time;
      tv1 : Int;
      tv2 : Int;
      tb1 : Bool;
      ti3 : Time;
      stabilizedelaytrigger : Bool;
      ti4 : Time;
      StabilizeTransition : Bool;
      StabilizeTransition_1 : Bool;
   END_VAR
BEGIN

REGION Network 1
   // Warmup Mode
         A     "SystemSTART_Pb";
         FP    #OS1;
         A     "IdleMode";
         S     "STARTSequnceBIT";

         CLR;
         A     "WarmupMode";
         JC    WormupMode;
         CLR;
         A     "StabilizeMode";
         JC    StabilizeMode;
         CLR;

         A     "GenerationMode";
         JC    GenerationMode;
         CLR;
         A     "CooldownMode";
         JC    CooldownMode;
         CLR;
         A     "IdleMode";
         JC    IdleMode;
         JU    EndOfLine;


   WormupMode:L     "WarmupRPM";
         T     "BafflePIDsp";
         L     "RPM";
         T     "BafflePIDin";

         SET;
         S     "OilPumpVFD_Ctrl";
         S     "Baffle_Ctrl";
         L     "WarmupVFDpct";
         T     "VFD_sp";

         L     "OilTemp";
         L     "WarmupOILTemp";
         >I;
         JC    WarmupTime;
         JU    StabilizeMode;


   WarmupTime:CALL  "CONVERTTIME"
         ( Int1 := "WarmupOilTempDelay_sp",
           tem1 := #ti1
         );
         CALL  TON, "IEC_Timer_0_DB_26"
         ( IN := TRUE,
           PT := #ti1,
           Q  := #warmupdelaytrigger,
           ET := #ti2
         );

         A     #warmupdelaytrigger;
         JC    WarmupExit;
         JU    StabilizeMode;

   WarmupExit:S     "WarmupTransition";
         CALL  RESET_TIMER
         ( "TIMER" := "IEC_Timer_0_DB_26"
         );

   // Stabilize Mode
   StabilizeMode:R     "WarmupTransition";
         L     "StabilizeKWsp";
         T     "BafflePIDsp";
         L     "Current";
         T     "BafflePIDin";
         L     "StabilizeKWsp";
         L     5;
         +I;
         T     #tv1;
         L     "StabilizeKWsp";
         L     5;
         -I;
         T     #tv2;
         L     "Current";
         L     #tv1;
         <I;
         S     #tb1;
         L     "Current";
         L     #tv2;
         >I;
         A     #tb1;
         JC    StabilizeTime;
         CALL  RESET_TIMER
         ( "TIMER" := "IEC_Timer_0_DB_27"
         );
         JU    GenerationMode;

   StabilizeTime:CALL  "CONVERTTIME"
         ( Int1 := "StabilizeDelay_sp",
           tem1 := #ti3
         );
         CALL  TON , "IEC_Timer_0_DB_27"
         ( IN := TRUE,
           PT := #ti3,
           Q  := #stabilizedelaytrigger,
           ET := #ti4
         );

         A     #stabilizedelaytrigger;
         JC    StabilizeExit;
         JU    GenerationMode;

   StabilizeExit:S     "StabilizeTransition";
         CALL  RESET_TIMER
         ( "TIMER" := "IEC_Timer_0_DB_26"
         );


   // Generation Mode
   GenerationMode:Rs;

   // Cooldown Mode
   CooldownMode:BE;


   // Idel Mode
   IdleMode:BE;


   // Fault Mode
   EndOfLine:BE;
END_REGION
END_FUNCTION_BLOCK

FUNCTION "SCP1" : Void   // FC1, FBD
{ S7_Optimized_Access := 'TRUE' }
VERSION : 0.1
   VAR_INPUT
      Input_Min : Int;
      Input_Signal : Int;
      Input_Max : Int;
      Output_Min : Int;
      Output_Max : Int;
   END_VAR
   VAR_OUTPUT
      SV : Int;
   END_VAR
   VAR_TEMP
      tv : Real;
   END_VAR
BEGIN

REGION Network 1
